C07270=1062.569,160.981,-81.280,172.441,30.431,155.615
C07271=1062.574,161.230,-81.303,172.443,30.435,155.616
C07272=1062.579,161.479,-81.325,172.445,30.437,155.616
C07273=1062.585,161.728,-81.347,172.446,30.440,155.616
C07274=1062.591,161.977,-81.369,172.448,30.443,155.617
C07275=1062.596,162.226,-81.392,172.450,30.446,155.617
C07276=1062.602,162.475,-81.413,172.453,30.449,155.618
C07277=1062.608,162.724,-81.436,172.454,30.452,155.618
C07278=1062.613,162.973,-81.458,172.456,30.455,155.619
C07279=1062.619,163.222,-81.480,172.458,30.458,155.619
C07280=1062.624,163.471,-81.503,172.460,30.461,155.620
C07281=1062.630,163.720,-81.525,172.461,30.463,155.620
C07282=1062.636,163.968,-81.547,172.463,30.466,155.621
C07283=1062.641,164.217,-81.569,172.465,30.469,155.621
C07284=1062.647,164.466,-81.592,172.468,30.472,155.622
C07285=1062.653,164.716,-81.614,172.469,30.475,155.622
C07286=1062.658,164.964,-81.636,172.471,30.478,155.622
C07287=1062.664,165.213,-81.659,172.473,30.481,155.623
C07288=1062.670,165.462,-81.681,172.475,30.484,155.623
C07289=1062.675,165.711,-81.703,172.476,30.487,155.624
C07290=1062.681,165.960,-81.726,172.478,30.490,155.624
C07291=1062.687,166.209,-81.747,172.480,30.492,155.625
C07292=1062.693,166.458,-81.770,172.483,30.496,155.625
C07293=1062.698,166.707,-81.793,172.484,30.498,155.626
C07294=1062.704,166.956,-81.815,172.486,30.501,155.626
C07295=1062.710,167.204,-81.837,172.488,30.504,155.627
C07296=1062.715,167.454,-81.860,172.490,30.507,155.627
C07297=1062.721,167.702,-81.883,172.491,30.510,155.627
C07298=1062.727,167.952,-81.904,172.494,30.513,155.628
C07299=1062.733,168.201,-81.927,172.496,30.516,155.628
C07300=1062.738,168.449,-81.950,172.498,30.519,155.629
C07301=1062.743,168.698,-81.972,172.499,30.521,155.629
C07302=1062.750,168.947,-81.994,172.501,30.524,155.630
C07303=1062.755,169.196,-82.017,172.503,30.527,155.630
C07304=1062.761,169.445,-82.040,172.506,30.530,155.631
C07305=1062.767,169.694,-82.062,172.507,30.533,155.631
C07306=1062.773,169.943,-82.084,172.509,30.536,155.632
C07307=1062.778,170.192,-82.107,172.511,30.539,155.632
C07308=1062.784,170.440,-82.130,172.513,30.541,155.632
C07309=1062.790,170.689,-82.152,172.514,30.545,155.633
C07310=1062.795,170.939,-82.174,172.517,30.547,155.633
C07311=1062.801,171.187,-82.197,172.519,30.551,155.634
C07312=1062.807,171.436,-82.220,172.521,30.553,155.634
C07313=1062.813,171.685,-82.243,172.523,30.556,155.635
C07314=1062.819,171.934,-82.265,172.524,30.559,155.635
C07315=1062.824,172.183,-82.288,172.526,30.562,155.636
C07316=1062.830,172.431,-82.310,172.529,30.565,155.636
C07317=1062.835,172.680,-82.333,172.531,30.568,155.637
C07318=1062.842,172.930,-82.355,172.532,30.571,155.637
C07319=1062.847,173.178,-82.378,172.534,30.573,155.637
C07320=1062.853,173.427,-82.401,172.536,30.576,155.638
C07321=1062.859,173.676,-82.424,172.539,30.579,155.638
C07322=1062.865,173.925,-82.446,172.540,30.582,155.639
C07323=1062.871,174.174,-82.469,172.542,30.585,155.639
C07324=1062.877,174.458,-82.494,172.545,30.589,155.640
C07325=1062.884,174.741,-82.521,172.547,30.592,155.640
C07326=1062.891,175.024,-82.547,172.549,30.595,155.641
C07327=1062.897,175.308,-82.572,172.551,30.598,155.641
C07328=1062.903,175.557,-82.595,172.553,30.601,155.642
C07329=1062.909,175.806,-82.618,172.556,30.604,155.642
C07330=1062.914,176.055,-82.641,172.557,30.607,155.643
C07331=1062.920,176.304,-82.664,172.559,30.610,155.643
C07332=1062.927,176.552,-82.686,172.561,30.612,155.644
C07333=1062.932,176.801,-82.709,172.564,30.616,155.644
C07334=1062.938,177.050,-82.732,172.565,30.618,155.645
C07335=1062.944,177.299,-82.755,172.567,30.621,155.645
C07336=1062.950,177.548,-82.778,172.569,30.624,155.646
C07337=1062.956,177.797,-82.800,172.572,30.627,155.646
C07338=1062.962,178.045,-82.823,172.573,30.630,155.646
C07339=1062.968,178.294,-82.846,172.575,30.633,155.647
C07340=1062.974,178.544,-82.869,172.577,30.636,155.647
C07341=1062.980,178.793,-82.892,172.580,30.638,155.648
C07342=1062.985,179.042,-82.915,172.581,30.642,155.648
C07343=1062.991,179.291,-82.938,172.583,30.644,155.649
C07344=1062.997,179.539,-82.961,172.585,30.647,155.649
C07345=1063.003,179.788,-82.984,172.588,30.650,155.650
C07346=1063.009,180.037,-83.007,172.590,30.653,155.650
C07347=1063.015,180.286,-83.029,172.591,30.656,155.651
C07348=1063.020,180.535,-83.052,172.593,30.659,155.651
C07349=1063.026,180.784,-83.075,172.596,30.662,155.651
C07350=1063.033,181.033,-83.099,172.598,30.665,155.652
C07351=1063.039,181.281,-83.122,172.599,30.667,155.652
C07352=1063.045,181.530,-83.145,172.601,30.670,155.653
C07353=1063.051,181.779,-83.168,172.604,30.673,155.653
C07354=1063.056,182.028,-83.191,172.606,30.676,155.654
C07355=1063.062,182.277,-83.214,172.607,30.679,155.654
C07356=1063.068,182.526,-83.236,172.610,30.682,155.655
C07357=1063.075,182.775,-83.261,172.612,30.685,155.655
C07358=1063.080,183.024,-83.283,172.614,30.687,155.655
C07359=1063.087,183.272,-83.306,172.615,30.691,155.656
C07360=1063.092,183.521,-83.329,172.618,30.693,155.656
C07361=1063.099,183.769,-83.352,172.620,30.696,155.657
C07362=1063.105,184.019,-83.376,172.622,30.699,155.657
C07363=1063.111,184.268,-83.399,172.625,30.702,155.658
C07364=1063.116,184.517,-83.422,172.626,30.705,155.658
C07365=1063.122,184.765,-83.445,172.628,30.708,155.659
C07366=1063.127,185.014,-83.469,172.631,30.711,155.659
C07367=1063.133,185.263,-83.492,172.633,30.714,155.660
C07368=1063.139,185.511,-83.515,172.634,30.717,155.660
C07369=1063.144,185.761,-83.539,172.636,30.720,155.661
C07370=1063.150,186.010,-83.562,172.639,30.723,155.661
C07371=1063.156,186.258,-83.586,172.641,30.726,155.662
C07372=1063.161,186.508,-83.609,172.642,30.730,155.662
C07373=1063.168,186.756,-83.633,172.645,30.732,155.663
C07374=1063.172,187.005,-83.657,172.647,30.736,155.663
C07375=1063.178,187.254,-83.680,172.649,30.739,155.664
C07376=1063.184,187.502,-83.703,172.650,30.742,155.664
C07377=1063.189,187.752,-83.727,172.653,30.745,155.665
C07378=1063.195,188.000,-83.750,172.655,30.748,155.665
C07379=1063.202,188.249,-83.774,172.657,30.751,155.666
C07380=1063.207,188.498,-83.798,172.659,30.754,155.666
C07381=1063.213,188.747,-83.821,172.661,30.757,155.666
C07382=1063.218,188.996,-83.845,172.663,30.760,155.667
C07383=1063.224,189.244,-83.868,172.666,30.763,155.667
C07384=1063.230,189.493,-83.892,172.668,30.766,155.668
C07385=1063.235,189.743,-83.916,172.669,30.769,155.668
C07386=1063.241,189.991,-83.939,172.672,30.773,155.669
C07387=1063.247,190.239,-83.964,172.674,30.775,155.669
C07388=1063.253,190.523,-83.990,172.677,30.779,155.670
C07389=1063.260,190.806,-84.017,172.678,30.782,155.671
C07390=1063.267,191.089,-84.043,172.681,30.786,155.671
C07391=1063.273,191.372,-84.071,172.684,30.789,155.672
C07392=1063.279,191.620,-84.094,172.686,30.792,155.672
C07393=1063.284,191.870,-84.118,172.687,30.795,155.673
C07394=1063.290,192.118,-84.142,172.690,30.798,155.673
C07395=1063.296,192.367,-84.166,172.692,30.801,155.674
C07396=1063.301,192.616,-84.189,172.694,30.805,155.674
C07397=1063.308,192.865,-84.213,172.696,30.807,155.675
C07398=1063.313,193.114,-84.238,172.698,30.811,155.675
C07399=1063.319,193.362,-84.260,172.700,30.814,155.676
C07400=1063.325,193.612,-84.285,172.703,30.817,155.676
C07401=1063.331,193.860,-84.309,172.704,30.820,155.677
C07402=1063.336,194.109,-84.332,172.707,30.823,155.677
C07403=1063.342,194.357,-84.356,172.709,30.826,155.678
C07404=1063.348,194.607,-84.381,172.711,30.829,155.678
C07405=1063.354,194.855,-84.404,172.714,30.832,155.679
C07406=1063.359,195.104,-84.428,172.715,30.835,155.679
C07407=1063.366,195.353,-84.452,172.717,30.838,155.680
C07408=1063.372,195.601,-84.475,172.720,30.842,155.680
C07409=1063.377,195.850,-84.500,172.722,30.844,155.680
C07410=1063.384,196.099,-84.524,172.724,30.848,155.681
C07411=1063.389,196.348,-84.547,172.726,30.851,155.682
C07412=1063.395,196.597,-84.571,172.728,30.853,155.682
C07413=1063.401,196.846,-84.596,172.731,30.857,155.682
C07414=1063.407,197.094,-84.619,172.732,30.860,155.683
C07415=1063.412,197.343,-84.643,172.735,30.863,155.683
C07416=1063.419,197.592,-84.668,172.737,30.866,155.684
C07417=1063.424,197.840,-84.692,172.739,30.869,155.684
C07418=1063.430,198.089,-84.716,172.742,30.872,155.685
C07419=1063.435,198.338,-84.739,172.743,30.875,155.685
C07420=1063.441,198.587,-84.763,172.746,30.879,155.686
C07421=1063.447,198.836,-84.788,172.748,30.881,155.686
C07422=1063.453,199.084,-84.811,172.751,30.884,155.687
C07423=1063.459,199.334,-84.836,172.752,30.888,155.687
C07424=1063.465,199.582,-84.860,172.754,30.891,155.688
C07425=1063.471,199.831,-84.884,172.757,30.894,155.688
C07426=1063.477,200.079,-84.908,172.759,30.897,155.689
C07427=1063.483,200.328,-84.932,172.761,30.900,155.689
C07428=1063.489,200.577,-84.956,172.763,30.903,155.690
C07429=1063.495,200.826,-84.980,172.766,30.906,155.690
C07430=1063.500,201.075,-85.005,172.768,30.909,155.691
C07431=1063.506,201.323,-85.029,172.770,30.912,155.691
C07432=1063.512,201.572,-85.053,172.772,30.915,155.692
C07433=1063.518,201.821,-85.077,172.774,30.919,155.692
C07434=1063.524,202.070,-85.102,172.777,30.921,155.693
C07435=1063.530,202.318,-85.125,172.779,30.925,155.693
C07436=1063.537,202.567,-85.151,172.781,30.928,155.694
C07437=1063.542,202.816,-85.175,172.783,30.931,155.694
C07438=1063.548,203.065,-85.199,172.786,30.934,155.695
C07439=1063.553,203.313,-85.224,172.788,30.938,155.695
C07440=1063.559,203.562,-85.247,172.790,30.941,155.696
C07441=1063.565,203.811,-85.272,172.792,30.944,155.697
C07442=1063.571,204.059,-85.297,172.794,30.947,155.697
C07443=1063.576,204.308,-85.322,172.797,30.950,155.697
C07444=1063.582,204.557,-85.346,172.799,30.953,155.698
C07445=1063.588,204.806,-85.370,172.801,30.957,155.699
C07446=1063.594,205.054,-85.394,172.803,30.960,155.699
C07447=1063.600,205.303,-85.419,172.806,30.963,155.700
C07448=1063.605,205.552,-85.444,172.808,30.966,155.700
C07449=1063.611,205.801,-85.468,172.811,30.970,155.701
C07450=1063.617,206.049,-85.493,172.812,30.973,155.701
C07451=1063.623,206.298,-85.518,172.815,30.976,155.702
C07452=1063.647,207.346,-85.621,172.981,31.057,155.708
C07453=1063.653,207.569,-85.644,172.982,31.060,155.709
C07454=1063.659,207.793,-85.667,172.984,31.064,155.710
C07455=1063.664,208.016,-85.689,172.986,31.068,155.710
C07456=1063.669,208.240,-85.712,172.988,31.071,155.711
C07457=1063.675,208.463,-85.735,172.988,31.075,155.712
C07458=1063.680,208.688,-85.758,172.990,31.079,155.712
C07459=1063.685,208.910,-85.781,172.992,31.082,155.713
C07460=1063.691,209.134,-85.804,172.994,31.086,155.714
C07461=1063.697,209.383,-85.829,172.996,31.090,155.714
C07462=1063.703,209.631,-85.854,172.998,31.094,155.715
C07463=1063.709,209.880,-85.880,173.000,31.098,155.716
C07464=1063.715,210.129,-85.906,173.002,31.102,155.717
C07465=1063.721,210.378,-85.931,173.004,31.106,155.717
C07466=1063.728,210.626,-85.957,173.006,31.111,155.718
C07467=1063.733,210.875,-85.983,173.008,31.114,155.719
C07468=1063.739,211.123,-86.008,173.010,31.119,155.720
C07469=1063.745,211.372,-86.034,173.012,31.122,155.720
C07470=1063.752,211.621,-86.059,173.014,31.127,155.721
C07471=1063.757,211.869,-86.085,173.016,31.131,155.722
C07472=1063.763,212.117,-86.111,173.018,31.135,155.722
C07473=1063.769,212.366,-86.136,173.020,31.139,155.723
C07474=1063.775,212.615,-86.162,173.022,31.143,155.724
C07475=1063.781,212.863,-86.187,173.024,31.147,155.725
C07476=1063.787,213.112,-86.213,173.026,31.151,155.725
C07477=1063.793,213.360,-86.239,173.027,31.155,155.726
C07478=1063.799,213.609,-86.265,173.030,31.159,155.727
C07479=1063.805,213.858,-86.290,173.032,31.164,155.728
C07480=1063.811,214.106,-86.317,173.034,31.167,155.728
C07481=1063.817,214.355,-86.342,173.036,31.172,155.729
C07482=1063.823,214.604,-86.368,173.037,31.175,155.730
C07483=1063.829,214.852,-86.393,173.040,31.180,155.730
C07484=1063.835,215.101,-86.420,173.042,31.184,155.731
C07485=1063.841,215.349,-86.445,173.044,31.188,155.732
C07486=1063.847,215.598,-86.472,173.045,31.192,155.733
C07487=1063.853,215.846,-86.497,173.048,31.196,155.733
C07488=1063.858,216.095,-86.523,173.050,31.200,155.734
C07489=1063.865,216.343,-86.549,173.052,31.204,155.735
C07490=1063.871,216.592,-86.574,173.054,31.208,155.736
C07491=1063.877,216.840,-86.601,173.056,31.212,155.736
C07492=1063.884,217.090,-86.627,173.058,31.216,155.737
C07493=1063.889,217.339,-86.653,173.060,31.220,155.738
C07494=1063.896,217.587,-86.679,173.062,31.225,155.738
C07495=1063.901,217.836,-86.705,173.064,31.228,155.739
C07496=1063.908,218.084,-86.731,173.066,31.233,155.740
C07497=1063.913,218.333,-86.757,173.068,31.236,155.741
C07498=1063.920,218.581,-86.783,173.070,31.240,155.741
C07499=1063.925,218.830,-86.809,173.072,31.244,155.742
C07500=1063.932,219.078,-86.835,173.074,31.248,155.743
C07501=1063.937,219.327,-86.861,173.077,31.253,155.743
C07502=1063.944,219.576,-86.887,173.079,31.256,155.744
C07503=1063.950,219.825,-86.913,173.080,31.261,155.745
C07504=1063.956,220.073,-86.939,173.083,31.264,155.746
C07505=1063.962,220.321,-86.966,173.085,31.268,155.746
C07506=1063.968,220.570,-86.991,173.087,31.272,155.747
C07507=1063.974,220.818,-87.018,173.088,31.276,155.748
C07508=1063.980,221.067,-87.043,173.091,31.281,155.748
C07509=1063.985,221.293,-87.067,173.093,31.284,155.749
C07510=1063.991,221.519,-87.091,173.095,31.287,155.750
C07511=1063.996,221.745,-87.115,173.097,31.291,155.750
C07512=1064.002,221.971,-87.139,173.098,31.295,155.751
C07513=1064.008,222.197,-87.163,173.100,31.299,155.752
C07514=1064.013,222.423,-87.187,173.102,31.302,155.752
C07515=1064.019,222.649,-87.211,173.104,31.306,155.753
C07516=1064.023,222.875,-87.235,173.106,31.310,155.754
C07517=1064.030,223.124,-87.262,173.108,31.314,155.754
C07518=1064.036,223.372,-87.288,173.110,31.318,155.755
C07519=1064.042,223.621,-87.314,173.112,31.322,155.756
C07520=1064.047,223.869,-87.340,173.115,31.326,155.757
C07521=1064.053,224.118,-87.367,173.116,31.330,155.757
C07522=1064.060,224.366,-87.393,173.118,31.334,155.758
C07523=1064.066,224.615,-87.420,173.121,31.338,155.759
C07524=1064.072,224.864,-87.446,173.123,31.342,155.759
C07525=1064.077,225.112,-87.473,173.125,31.346,155.760
C07526=1064.084,225.360,-87.499,173.127,31.350,155.761
C07527=1064.090,225.608,-87.525,173.129,31.354,155.762
C07528=1064.096,225.857,-87.552,173.131,31.358,155.762
C07529=1064.102,226.106,-87.579,173.134,31.362,155.763
C07530=1064.107,226.355,-87.605,173.135,31.366,155.764
C07531=1064.114,226.603,-87.631,173.137,31.370,155.764
C07532=1064.120,226.852,-87.658,173.140,31.374,155.765
C07533=1064.126,227.100,-87.685,173.142,31.378,155.766
C07534=1064.132,227.349,-87.711,173.145,31.382,155.767
C07535=1064.137,227.597,-87.738,173.146,31.386,155.767
C07536=1064.145,227.846,-87.764,173.148,31.390,155.768
C07537=1064.150,228.094,-87.791,173.151,31.394,155.769
C07538=1064.156,228.342,-87.818,173.153,31.398,155.769
C07539=1064.163,228.592,-87.845,173.154,31.402,155.770
C07540=1064.168,228.840,-87.871,173.157,31.406,155.771
C07541=1064.175,229.088,-87.898,173.159,31.409,155.772
C07542=1064.181,229.337,-87.925,173.161,31.414,155.772
C07543=1064.187,229.585,-87.951,173.164,31.417,155.773
C07544=1064.193,229.834,-87.978,173.165,31.422,155.774
C07545=1064.199,230.083,-88.005,173.168,31.426,155.774
C07546=1064.205,230.331,-88.031,173.170,31.429,155.775
C07547=1064.211,230.580,-88.058,173.172,31.434,155.776
C07548=1064.216,230.828,-88.085,173.175,31.437,155.777
C07549=1064.223,231.076,-88.113,173.176,31.442,155.777
C07550=1064.229,231.325,-88.139,173.179,31.445,155.778
C07551=1064.235,231.573,-88.166,173.181,31.450,155.779
C07552=1064.241,231.822,-88.193,173.183,31.453,155.779
C07553=1064.247,232.070,-88.219,173.186,31.457,155.780
C07554=1064.253,232.319,-88.246,173.187,31.462,155.781
C07555=1064.259,232.567,-88.274,173.189,31.465,155.782
C07556=1064.265,232.816,-88.300,173.192,31.470,155.782
C07557=1064.271,233.064,-88.327,173.194,31.473,155.783
C07558=1064.277,233.313,-88.354,173.197,31.477,155.784
C07559=1064.283,233.561,-88.381,173.198,31.481,155.784
C07560=1064.289,233.810,-88.409,173.200,31.485,155.785
C07561=1064.295,234.059,-88.436,173.203,31.490,155.786
C07562=1064.300,234.307,-88.462,173.205,31.493,155.787
C07563=1064.307,234.555,-88.490,173.208,31.498,155.787
C07564=1064.313,234.804,-88.517,173.209,31.501,155.788
C07565=1064.318,235.026,-88.541,173.211,31.505,155.789
C07566=1064.323,235.248,-88.565,173.213,31.508,155.789
C07567=1064.329,235.470,-88.590,173.216,31.512,155.790
C07568=1064.334,235.691,-88.614,173.218,31.516,155.791
C07569=1064.340,235.914,-88.638,173.219,31.519,155.791
C07570=1064.345,236.136,-88.663,173.221,31.523,155.792
C07571=1064.351,236.358,-88.687,173.223,31.526,155.792
C07572=1064.356,236.580,-88.711,173.225,31.530,155.793
C07573=1064.361,236.828,-88.738,173.228,31.534,155.794
C07574=1064.368,237.077,-88.765,173.230,31.538,155.795
C07575=1064.374,237.325,-88.793,173.232,31.542,155.795
C07576=1064.380,237.574,-88.820,173.234,31.545,155.796
C07577=1064.386,237.822,-88.847,173.237,31.550,155.797
C07578=1064.392,238.071,-88.874,173.239,31.554,155.797
C07579=1064.398,238.319,-88.902,173.242,31.557,155.798
C07580=1064.404,238.568,-88.929,173.243,31.562,155.799
C07581=1064.410,238.816,-88.956,173.245,31.565,155.800
C07582=1064.416,239.065,-88.984,173.248,31.569,155.800
C07583=1064.422,239.313,-89.011,173.250,31.573,155.801
C07584=1064.429,239.562,-89.038,173.253,31.577,155.802
C07585=1064.435,239.809,-89.066,173.254,31.581,155.802
C07586=1064.441,240.058,-89.094,173.257,31.585,155.803
C07587=1064.446,240.307,-89.121,173.259,31.589,155.804
C07588=1064.453,240.555,-89.148,173.262,31.593,155.805
C07589=1064.458,240.804,-89.176,173.264,31.597,155.805
C07590=1064.465,241.052,-89.203,173.267,31.601,155.806
C07591=1064.471,241.300,-89.231,173.268,31.605,155.807
C07592=1064.477,241.549,-89.258,173.271,31.609,155.807
C07593=1064.483,241.797,-89.286,173.273,31.613,155.808
C07594=1064.489,242.045,-89.313,173.276,31.617,155.809
C07595=1064.495,242.294,-89.340,173.278,31.621,155.809
C07596=1064.501,242.542,-89.368,173.280,31.625,155.810
C07597=1064.508,242.791,-89.396,173.282,31.629,155.811
C07598=1064.513,243.040,-89.423,173.284,31.632,155.812
C07599=1064.519,243.288,-89.451,173.287,31.636,155.812
C07600=1064.525,243.536,-89.479,173.289,31.641,155.813
C07601=1064.531,243.785,-89.507,173.292,31.644,155.814
C07602=1064.537,244.033,-89.535,173.293,31.649,155.815
C07603=1064.543,244.282,-89.562,173.296,31.652,155.815
C07604=1064.548,244.530,-89.590,173.298,31.657,155.816
C07605=1064.555,244.778,-89.617,173.301,31.660,155.817
C07606=1064.560,245.026,-89.645,173.303,31.664,155.817
C07607=1064.567,245.275,-89.673,173.305,31.669,155.818
C07608=1064.573,245.523,-89.701,173.307,31.672,155.819
C07609=1064.579,245.771,-89.729,173.310,31.676,155.819
C07610=1064.585,246.021,-89.756,173.312,31.680,155.820
C07611=1064.591,246.268,-89.784,173.315,31.684,155.821
C07612=1064.597,246.517,-89.812,173.317,31.688,155.822
C07613=1064.603,246.766,-89.840,173.319,31.692,155.822
C07614=1064.609,247.013,-89.868,173.322,31.696,155.823
C07615=1064.615,247.262,-89.896,173.324,31.700,155.824
C07616=1064.620,247.510,-89.924,173.327,31.704,155.824
C07617=1064.626,247.759,-89.952,173.329,31.708,155.825
C07618=1064.633,248.007,-89.980,173.332,31.712,155.826
C07619=1064.638,248.256,-90.008,173.333,31.716,155.827
C07620=1064.644,248.504,-90.036,173.336,31.720,155.827
C07621=1064.649,248.723,-90.061,173.338,31.724,155.828
C07622=1064.654,248.942,-90.086,173.340,31.727,155.829
C07623=1064.660,249.161,-90.111,173.342,31.731,155.829
C07624=1064.665,249.380,-90.136,173.345,31.734,155.830
C07625=1064.670,249.599,-90.160,173.346,31.738,155.831
C07626=1064.675,249.818,-90.185,173.348,31.741,155.831
C07627=1064.681,250.036,-90.210,173.350,31.745,155.832
C07628=1064.686,250.255,-90.235,173.352,31.748,155.833
C07629=1064.692,250.502,-90.263,173.355,31.752,155.833
C07630=1064.698,250.751,-90.291,173.358,31.757,155.834
C07631=1064.704,251.000,-90.319,173.360,31.760,155.835
C07632=1064.709,251.248,-90.347,173.362,31.764,155.835
C07633=1064.715,251.497,-90.376,173.364,31.768,155.836
C07634=1064.722,251.745,-90.403,173.367,31.772,155.837
C07635=1064.728,251.993,-90.432,173.369,31.776,155.838
C07636=1064.734,252.241,-90.460,173.372,31.780,155.838
C07637=1064.739,252.490,-90.489,173.375,31.784,155.839
C07638=1064.745,252.739,-90.517,173.376,31.788,155.840
C07639=1064.752,252.986,-90.545,173.379,31.792,155.840
C07640=1064.758,253.235,-90.573,173.381,31.796,155.841
C07641=1064.764,253.483,-90.602,173.384,31.800,155.842
C07642=1064.770,253.732,-90.631,173.386,31.804,155.843
C07643=1064.775,253.980,-90.659,173.389,31.808,155.843
C07644=1064.782,254.228,-90.687,173.391,31.812,155.844
C07645=1064.788,254.476,-90.716,173.393,31.816,155.845
C07646=1064.794,254.725,-90.744,173.396,31.820,155.845
C07647=1064.800,254.973,-90.772,173.398,31.823,155.846
C07648=1064.806,255.221,-90.801,173.401,31.828,155.847
C07649=1064.812,255.470,-90.829,173.404,31.832,155.848
C07650=1064.819,255.718,-90.858,173.406,31.835,155.848
C07651=1064.825,255.966,-90.886,173.408,31.840,155.849
C07652=1064.830,256.214,-90.915,173.410,31.843,155.850
C07653=1064.836,256.463,-90.943,173.413,31.847,155.850
C07654=1064.842,256.711,-90.971,173.416,31.851,155.851
C07655=1064.848,256.960,-91.000,173.418,31.855,155.852
C07656=1064.854,257.208,-91.029,173.421,31.859,155.853
C07657=1064.861,257.456,-91.057,173.422,31.863,155.853
C07658=1064.867,257.705,-91.085,173.425,31.867,155.854
C07659=1064.873,257.952,-91.114,173.428,31.871,155.855
C07660=1064.879,258.200,-91.143,173.430,31.875,155.855
C07661=1064.885,258.449,-91.171,173.433,31.879,155.856
C07662=1064.891,258.697,-91.201,173.436,31.883,155.857
C07663=1064.897,258.946,-91.229,173.438,31.887,155.858
C07664=1064.904,259.194,-91.258,173.440,31.891,155.858
C07665=1064.910,259.443,-91.286,173.443,31.894,155.859
C07666=1064.917,259.691,-91.315,173.445,31.898,155.860
C07667=1064.923,259.939,-91.344,173.448,31.902,155.860
C07668=1064.929,260.188,-91.372,173.450,31.906,155.861
C07669=1064.935,260.436,-91.401,173.453,31.910,155.862
C07670=1064.941,260.684,-91.430,173.456,31.914,155.863
C07671=1064.947,260.932,-91.458,173.457,31.918,155.863
C07672=1064.953,261.180,-91.487,173.460,31.922,155.864
C07673=1064.959,261.428,-91.516,173.463,31.926,155.865
C07674=1064.965,261.676,-91.545,173.465,31.929,155.865
C07675=1064.971,261.925,-91.574,173.468,31.933,155.866
C07676=1064.977,262.173,-91.603,173.471,31.938,155.867
C07677=1064.984,262.391,-91.627,173.473,31.941,155.867
C07678=1064.989,262.609,-91.653,173.475,31.944,155.868
C07679=1064.994,262.827,-91.678,173.477,31.948,155.869
C07680=1065.000,263.045,-91.704,173.479,31.951,155.869
C07681=1065.006,263.262,-91.729,173.482,31.954,155.870
C07682=1065.011,263.480,-91.754,173.484,31.958,155.871
C07683=1065.016,263.698,-91.780,173.486,31.961,155.871
C07684=1065.022,263.915,-91.806,173.489,31.965,155.872
C07685=1065.028,264.164,-91.834,173.491,31.969,155.872
C07686=1065.033,264.412,-91.864,173.493,31.973,155.873
C07687=1065.040,264.661,-91.893,173.496,31.977,155.874
C07688=1065.045,264.908,-91.921,173.498,31.981,155.875
C07689=1065.052,265.156,-91.950,173.501,31.985,155.875
C07690=1065.057,265.405,-91.980,173.504,31.989,155.876
C07691=1065.063,265.653,-92.009,173.506,31.993,155.877
C07692=1065.070,265.901,-92.038,173.509,31.996,155.878
C07693=1065.076,266.149,-92.067,173.511,32.001,155.878
C07694=1065.081,266.397,-92.097,173.514,32.005,155.879
C07695=1065.088,266.645,-92.126,173.516,32.009,155.880
C07696=1065.094,266.894,-92.155,173.519,32.012,155.880
C07697=1065.100,267.143,-92.185,173.522,32.017,155.881
C07698=1065.106,267.391,-92.214,173.524,32.020,155.882
C07699=1065.112,267.639,-92.243,173.527,32.024,155.883
C07700=1065.119,267.887,-92.273,173.530,32.029,155.883
C07701=1065.125,268.135,-92.302,173.531,32.032,155.884
C07702=1065.131,268.383,-92.331,173.534,32.037,155.885
C07703=1065.137,268.631,-92.360,173.537,32.040,155.886
C07704=1065.143,268.880,-92.390,173.540,32.044,155.886
C07705=1065.149,269.128,-92.419,173.542,32.048,155.887
C07706=1065.155,269.376,-92.448,173.545,32.052,155.888
C07707=1065.161,269.624,-92.479,173.548,32.056,155.888
C07708=1065.167,269.872,-92.508,173.551,32.060,155.889
C07709=1065.173,270.120,-92.537,173.552,32.064,155.890
C07710=1065.179,270.369,-92.567,173.555,32.068,155.891
C07711=1065.185,270.617,-92.597,173.558,32.072,155.891
C07712=1065.192,270.865,-92.626,173.561,32.076,155.892
C07713=1065.198,271.113,-92.655,173.563,32.080,155.893
C07714=1065.203,271.362,-92.685,173.566,32.084,155.894
C07715=1065.210,271.609,-92.714,173.569,32.088,155.894
C07716=1065.215,271.858,-92.744,173.572,32.092,155.895
C07717=1065.222,272.105,-92.774,173.573,32.096,155.896
C07718=1065.228,272.354,-92.804,173.576,32.100,155.897
C07719=1065.234,272.602,-92.833,173.579,32.104,155.897
C07720=1065.240,272.850,-92.863,173.582,32.108,155.898
C07721=1065.246,273.098,-92.892,173.584,32.112,155.899
C07722=1065.252,273.347,-92.922,173.587,32.116,155.899
C07723=1065.258,273.594,-92.952,173.590,32.120,155.900
C07724=1065.264,273.843,-92.981,173.593,32.124,155.901
C07725=1065.271,274.091,-93.011,173.594,32.128,155.902
C07726=1065.277,274.339,-93.041,173.597,32.132,155.902
C07727=1065.282,274.587,-93.071,173.600,32.136,155.903
C07728=1065.289,274.835,-93.100,173.603,32.140,155.904
C07729=1065.294,275.083,-93.131,173.606,32.144,155.905
C07730=1065.301,275.332,-93.160,173.608,32.148,155.905
C07731=1065.307,275.580,-93.191,173.611,32.152,155.906
C07732=1065.313,275.828,-93.221,173.614,32.156,155.907
C07733=1065.318,276.048,-93.247,173.616,32.160,155.908
C07734=1065.323,276.267,-93.273,173.618,32.163,155.908
C07735=1065.329,276.487,-93.300,173.620,32.167,155.909
C07736=1065.335,276.706,-93.326,173.623,32.170,155.909
C07737=1065.340,276.925,-93.353,173.625,32.174,155.910
C07738=1065.346,277.145,-93.379,173.628,32.178,155.911
C07739=1065.350,277.364,-93.406,173.630,32.181,155.911
C07740=1065.356,277.584,-93.433,173.633,32.185,155.912
C07741=1065.362,277.832,-93.462,173.636,32.189,155.913
C07742=1065.368,278.080,-93.493,173.638,32.192,155.914
C07743=1065.374,278.328,-93.523,173.641,32.197,155.914
C07744=1065.380,278.577,-93.553,173.643,32.201,155.915
C07745=1065.387,278.825,-93.583,173.646,32.205,155.916
C07746=1065.393,279.073,-93.613,173.649,32.209,155.916
C07747=1065.399,279.321,-93.644,173.651,32.213,155.917
C07748=1065.405,279.569,-93.673,173.654,32.217,155.918
C07749=1065.411,279.817,-93.703,173.657,32.221,155.919
C07750=1065.417,280.066,-93.734,173.660,32.225,155.920
C07751=1065.423,280.313,-93.764,173.663,32.229,155.920
C07752=1065.429,280.561,-93.795,173.666,32.233,155.921
C07753=1065.436,280.809,-93.824,173.667,32.237,155.922
C07754=1065.442,281.058,-93.854,173.670,32.241,155.923
C07755=1065.448,281.306,-93.885,173.673,32.245,155.923
C07756=1065.453,281.553,-93.915,173.676,32.249,155.924
C07757=1065.460,281.802,-93.946,173.679,32.253,155.925
C07758=1065.466,282.050,-93.976,173.682,32.258,155.926
C07759=1065.471,282.298,-94.007,173.684,32.261,155.926
C07760=1065.478,282.546,-94.037,173.687,32.266,155.927
C07761=1065.484,282.794,-94.068,173.690,32.269,155.928
C07762=1065.489,283.042,-94.098,173.693,32.274,155.929
C07763=1065.496,283.290,-94.129,173.695,32.278,155.929
C07764=1065.502,283.538,-94.159,173.698,32.282,155.930
C07765=1065.508,283.786,-94.189,173.701,32.286,155.931
C07766=1065.514,284.034,-94.220,173.704,32.290,155.932
C07767=1065.520,284.282,-94.250,173.706,32.294,155.932
C07768=1065.526,284.531,-94.281,173.709,32.298,155.933
C07769=1065.532,284.778,-94.312,173.712,32.302,155.934
C07770=1065.539,285.026,-94.342,173.715,32.306,155.935
C07771=1065.545,285.274,-94.373,173.718,32.310,155.935
C07772=1065.551,285.522,-94.403,173.721,32.314,155.936
C07773=1065.558,285.770,-94.434,173.724,32.318,155.937
C07774=1065.563,286.018,-94.464,173.726,32.323,155.938
C07775=1065.570,286.266,-94.496,173.728,32.326,155.938
C07776=1065.576,286.514,-94.526,173.731,32.331,155.939
C07777=1065.582,286.762,-94.556,173.734,32.335,155.940
C07778=1065.588,287.010,-94.587,173.737,32.339,155.941
C07779=1065.594,287.258,-94.617,173.740,32.343,155.941
C07780=1065.601,287.506,-94.649,173.743,32.347,155.942
C07781=1065.606,287.754,-94.679,173.746,32.351,155.943
C07782=1065.613,288.002,-94.710,173.749,32.355,155.944
C07783=1065.619,288.250,-94.741,173.752,32.359,155.945
C07784=1065.625,288.498,-94.772,173.755,32.363,155.945
C07785=1065.631,288.746,-94.803,173.757,32.367,155.946
C07786=1065.637,288.994,-94.834,173.760,32.372,155.947
C07787=1065.643,289.242,-94.864,173.762,32.375,155.947
C07788=1065.649,289.490,-94.895,173.765,32.380,155.948
C07789=1065.654,289.715,-94.923,173.768,32.383,155.949
C07790=1065.661,289.940,-94.951,173.771,32.387,155.950
C07791=1065.666,290.165,-94.980,173.773,32.391,155.950
C07792=1065.672,290.389,-95.007,173.776,32.394,155.951
C07793=1065.677,290.614,-95.036,173.779,32.399,155.952
C07794=1065.683,290.839,-95.064,173.781,32.402,155.953
C07795=1065.688,291.063,-95.092,173.784,32.406,155.953
C07796=1065.694,291.288,-95.121,173.787,32.410,155.954
C07797=1065.700,291.536,-95.151,173.789,32.414,155.955
C07798=1065.706,291.784,-95.182,173.792,32.418,155.955
C07799=1065.712,292.032,-95.213,173.795,32.422,155.956
C07800=1065.718,292.280,-95.245,173.798,32.426,155.957
C07801=1065.725,292.529,-95.276,173.801,32.430,155.958
C07802=1065.731,292.776,-95.307,173.803,32.435,155.959
C07803=1065.737,293.024,-95.339,173.806,32.438,155.959
C07804=1065.743,293.272,-95.369,173.809,32.443,155.960
C07805=1065.749,293.520,-95.400,173.812,32.447,155.961
C07806=1065.755,293.768,-95.432,173.815,32.451,155.962
C07807=1065.761,294.016,-95.463,173.818,32.455,155.962
C07808=1065.768,294.264,-95.494,173.821,32.459,155.963
C07809=1065.774,294.511,-95.525,173.824,32.463,155.964
C07810=1065.780,294.760,-95.557,173.827,32.468,155.965
C07811=1065.786,295.008,-95.588,173.829,32.472,155.966
C07812=1065.792,295.255,-95.620,173.832,32.476,155.966
C07813=1065.799,295.503,-95.651,173.835,32.480,155.967
C07814=1065.805,295.752,-95.682,173.838,32.484,155.968
C07815=1065.810,295.999,-95.714,173.841,32.488,155.969
C07816=1065.817,296.247,-95.745,173.844,32.493,155.969
C07817=1065.823,296.495,-95.777,173.847,32.497,155.970
C07818=1065.829,296.742,-95.808,173.850,32.501,155.971
C07819=1065.835,296.991,-95.840,173.853,32.505,155.972
C07820=1065.842,297.239,-95.871,173.856,32.510,155.973
C07821=1065.847,297.487,-95.902,173.859,32.514,155.974
C07822=1065.854,297.735,-95.934,173.862,32.518,155.974
C07823=1065.860,297.983,-95.966,173.865,32.522,155.975
C07824=1065.865,298.230,-95.998,173.868,32.527,155.976
C07825=1065.872,298.478,-96.029,173.871,32.531,155.977
C07826=1065.878,298.726,-96.061,173.873,32.535,155.978
C07827=1065.883,298.974,-96.093,173.876,32.539,155.978
C07828=1065.889,299.222,-96.125,173.879,32.544,155.979
C07829=1065.896,299.470,-96.156,173.882,32.548,155.980
C07830=1065.902,299.717,-96.189,173.885,32.552,155.981
C07831=1065.908,299.965,-96.221,173.888,32.556,155.982
C07832=1065.914,300.213,-96.252,173.891,32.561,155.982
C07833=1065.920,300.461,-96.284,173.895,32.565,155.983
C07834=1065.926,300.709,-96.316,173.898,32.569,155.984
C07835=1065.932,300.957,-96.348,173.901,32.574,155.985
C07836=1065.938,301.205,-96.379,173.904,32.578,155.986
C07837=1065.944,301.452,-96.411,173.907,32.583,155.987
C07838=1065.950,301.700,-96.444,173.910,32.587,155.987
C07839=1065.956,301.948,-96.476,173.913,32.591,155.988
C07840=1065.963,302.196,-96.507,173.916,32.595,155.989
C07841=1065.968,302.444,-96.539,173.919,32.600,155.990
C07842=1065.974,302.691,-96.571,173.922,32.604,155.991
C07843=1065.980,302.939,-96.603,173.924,32.608,155.991
C07844=1065.987,303.187,-96.635,173.927,32.612,155.992
C07845=1065.993,303.419,-96.665,173.930,32.617,155.993
C07846=1065.998,303.651,-96.695,173.933,32.620,155.994
C07847=1066.004,303.884,-96.725,173.936,32.624,155.994
C07848=1066.010,304.116,-96.755,173.939,32.629,155.995
C07849=1066.016,304.349,-96.786,173.942,32.632,155.996
C07850=1066.021,304.581,-96.815,173.945,32.637,155.997
C07851=1066.027,304.813,-96.845,173.947,32.641,155.998
C07852=1066.033,305.045,-96.875,173.950,32.644,155.998
C07853=1066.039,305.293,-96.908,173.953,32.649,155.999
C07854=1066.045,305.541,-96.940,173.957,32.654,156.000
C07855=1066.051,305.789,-96.973,173.960,32.658,156.001
C07856=1066.058,306.037,-97.004,173.963,32.662,156.002
C07857=1066.064,306.284,-97.037,173.966,32.666,156.002
C07858=1066.070,306.533,-97.069,173.969,32.670,156.003
C07859=1066.076,306.779,-97.101,173.972,32.675,156.004
C07860=1066.082,307.028,-97.133,173.975,32.679,156.005
C07861=1066.089,307.275,-97.166,173.978,32.683,156.006
C07862=1066.095,307.523,-97.198,173.982,32.688,156.007
C07863=1066.101,307.771,-97.230,173.985,32.692,156.007
C07864=1066.107,308.019,-97.262,173.988,32.697,156.008
C07865=1066.114,308.267,-97.295,173.990,32.701,156.009
C07866=1066.120,308.514,-97.328,173.993,32.705,156.010
C07867=1066.127,308.762,-97.359,173.996,32.709,156.011
C07868=1066.133,309.010,-97.392,173.999,32.713,156.011
C07869=1066.139,309.258,-97.424,174.003,32.718,156.012
C07870=1066.145,309.505,-97.457,174.006,32.723,156.013
C07871=1066.151,309.753,-97.489,174.009,32.727,156.014
C07872=1066.158,310.001,-97.522,174.012,32.731,156.015
C07873=1066.164,310.249,-97.554,174.015,32.735,156.016
C07874=1066.170,310.496,-97.587,174.018,32.740,156.017
C07875=1066.177,310.744,-97.619,174.022,32.744,156.017
C07876=1066.184,310.992,-97.652,174.025,32.749,156.018
C07877=1066.190,311.240,-97.684,174.028,32.753,156.019
C07878=1066.196,311.488,-97.717,174.031,32.757,156.020
C07879=1066.203,311.735,-97.750,174.034,32.761,156.021
C07880=1066.209,311.983,-97.783,174.038,32.766,156.022
C07881=1066.215,312.231,-97.815,174.041,32.770,156.022
C07882=1066.221,312.479,-97.847,174.044,32.775,156.023
C07883=1066.227,312.726,-97.880,174.047,32.779,156.024
C07884=1066.234,312.975,-97.913,174.050,32.783,156.025
C07885=1066.241,313.222,-97.946,174.054,32.788,156.026
C07886=1066.247,313.470,-97.979,174.057,32.792,156.027
C07887=1066.254,313.717,-98.011,174.060,32.796,156.027
C07888=1066.260,313.965,-98.044,174.063,32.800,156.028
C07889=1066.266,314.213,-98.077,174.066,32.805,156.029
C07890=1066.272,314.460,-98.110,174.070,32.810,156.030
C07891=1066.278,314.708,-98.142,174.073,32.814,156.031
C07892=1066.284,314.956,-98.176,174.076,32.819,156.032
C07893=1066.291,315.204,-98.209,174.079,32.823,156.033
C07894=1066.296,315.452,-98.242,174.082,32.828,156.034
C07895=1066.303,315.700,-98.275,174.086,32.832,156.034
C07896=1066.309,315.947,-98.308,174.089,32.837,156.035
C07897=1066.315,316.194,-98.342,174.092,32.841,156.036
C07898=1066.321,316.442,-98.374,174.095,32.846,156.037
C07899=1066.327,316.690,-98.408,174.098,32.851,156.038
C07900=1066.333,316.938,-98.440,174.102,32.855,156.039
C07901=1066.339,317.171,-98.472,174.105,32.859,156.040
C07902=1066.345,317.406,-98.504,174.108,32.864,156.041
C07903=1066.350,317.640,-98.535,174.111,32.868,156.041
C07904=1066.357,317.874,-98.567,174.114,32.872,156.042
C07905=1066.362,318.109,-98.598,174.117,32.877,156.043
C07906=1066.368,318.342,-98.629,174.120,32.881,156.044
C07907=1066.374,318.576,-98.661,174.123,32.886,156.045
C07908=1066.380,318.811,-98.693,174.126,32.890,156.046
C07909=1066.386,319.058,-98.726,174.128,32.894,156.046
C07910=1066.392,319.306,-98.759,174.132,32.899,156.047
C07911=1066.398,319.554,-98.792,174.135,32.904,156.048
C07912=1066.405,319.802,-98.826,174.138,32.908,156.049
C07913=1066.411,320.049,-98.859,174.141,32.913,156.050
C07914=1066.417,320.297,-98.893,174.145,32.917,156.051
C07915=1066.423,320.544,-98.926,174.148,32.922,156.052
C07916=1066.429,320.793,-98.960,174.151,32.926,156.053
C07917=1066.436,321.040,-98.993,174.154,32.931,156.054
C07918=1066.441,321.288,-99.027,174.158,32.935,156.054
C07919=1066.448,321.535,-99.060,174.161,32.940,156.055
C07920=1066.454,321.783,-99.094,174.164,32.945,156.056
C07921=1066.461,322.030,-99.127,174.168,32.949,156.057
C07922=1066.467,322.279,-99.161,174.171,32.954,156.058
C07923=1066.473,322.526,-99.194,174.174,32.959,156.059
C07924=1066.479,322.773,-99.228,174.177,32.963,156.060
C07925=1066.486,323.021,-99.261,174.181,32.968,156.061
C07926=1066.492,323.269,-99.296,174.185,32.972,156.062
C07927=1066.498,323.516,-99.328,174.188,32.977,156.063
C07928=1066.505,323.764,-99.363,174.192,32.982,156.064
C07929=1066.511,324.011,-99.396,174.195,32.986,156.064
C07930=1066.518,324.260,-99.430,174.198,32.991,156.065
C07931=1066.523,324.507,-99.464,174.202,32.996,156.066
C07932=1066.531,324.755,-99.498,174.205,33.000,156.067
C07933=1066.536,325.003,-99.531,174.208,33.005,156.068
C07934=1066.543,325.250,-99.565,174.212,33.009,156.069
C07935=1066.549,325.498,-99.599,174.215,33.014,156.070
C07936=1066.556,325.745,-99.632,174.218,33.019,156.071
C07937=1066.562,325.993,-99.667,174.222,33.024,156.072
C07938=1066.568,326.240,-99.700,174.225,33.028,156.073
C07939=1066.575,326.488,-99.734,174.228,33.033,156.074
C07940=1066.581,326.736,-99.768,174.232,33.037,156.075
C07941=1066.588,326.983,-99.802,174.235,33.042,156.075
C07942=1066.595,327.231,-99.836,174.238,33.047,156.076
C07943=1066.600,327.478,-99.870,174.242,33.052,156.077
C07944=1066.608,327.726,-99.904,174.245,33.056,156.078
C07945=1066.613,327.974,-99.938,174.249,33.061,156.079
C07946=1066.620,328.222,-99.971,174.252,33.065,156.080
C07947=1066.626,328.469,-100.005,174.255,33.070,156.081
C07948=1066.633,328.717,-100.040,174.259,33.075,156.082
C07949=1066.640,328.965,-100.074,174.262,33.080,156.083
C07950=1066.646,329.212,-100.108,174.266,33.085,156.084
C07951=1066.652,329.460,-100.142,174.269,33.089,156.085
C07952=1066.659,329.707,-100.176,174.272,33.094,156.086
C07953=1066.665,329.955,-100.210,174.276,33.099,156.087
C07954=1066.672,330.202,-100.245,174.279,33.103,156.088
C07955=1066.679,330.449,-100.279,174.283,33.108,156.089
C07956=1066.685,330.697,-100.313,174.286,33.113,156.089
C07957=1066.691,330.929,-100.344,174.289,33.117,156.090
C07958=1066.697,331.160,-100.377,174.292,33.122,156.091
C07959=1066.703,331.391,-100.409,174.296,33.126,156.092
C07960=1066.708,331.621,-100.441,174.299,33.131,156.093
C07961=1066.715,331.853,-100.473,174.302,33.136,156.094
C07962=1066.721,332.084,-100.505,174.305,33.140,156.095
C07963=1066.726,332.315,-100.538,174.308,33.144,156.096
C07964=1066.732,332.547,-100.570,174.312,33.149,156.097
C07965=1066.738,332.794,-100.604,174.315,33.154,156.098
C07966=1066.745,333.041,-100.639,174.318,33.159,156.099
C07967=1066.751,333.289,-100.674,174.323,33.164,156.100
C07968=1066.757,333.536,-100.708,174.326,33.169,156.101
C07969=1066.764,333.784,-100.743,174.330,33.173,156.102
C07970=1066.771,334.032,-100.777,174.333,33.178,156.102
C07971=1066.776,334.279,-100.811,174.337,33.184,156.104
C07972=1066.783,334.526,-100.847,174.340,33.188,156.104
C07973=1066.790,334.774,-100.881,174.344,33.193,156.105
C07974=1066.796,335.022,-100.916,174.347,33.198,156.106
C07975=1066.802,335.269,-100.950,174.351,33.203,156.107
C07976=1066.809,335.516,-100.985,174.354,33.208,156.108
C07977=1066.816,335.764,-101.020,174.358,33.213,156.109
C07978=1066.822,336.012,-101.055,174.361,33.218,156.110
C07979=1066.828,336.259,-101.089,174.365,33.223,156.111
C07980=1066.835,336.506,-101.124,174.368,33.228,156.112
C07981=1066.842,336.754,-101.159,174.371,33.232,156.113
C07982=1066.848,337.002,-101.194,174.375,33.238,156.114
C07983=1066.855,337.249,-101.229,174.379,33.243,156.115
C07984=1066.860,337.497,-101.263,174.382,33.248,156.116
C07985=1066.867,337.744,-101.299,174.385,33.253,156.117
C07986=1066.874,337.991,-101.334,174.390,33.258,156.118
C07987=1066.880,338.239,-101.368,174.394,33.263,156.119
C07988=1066.886,338.487,-101.404,174.397,33.268,156.121
C07989=1066.892,338.734,-101.439,174.401,33.273,156.121
C07990=1066.899,338.981,-101.474,174.404,33.278,156.123
C07991=1066.906,339.229,-101.509,174.408,33.283,156.124
C07992=1066.911,339.477,-101.544,174.411,33.288,156.125
C07993=1066.918,339.724,-101.579,174.415,33.293,156.126
C07994=1066.925,339.972,-101.614,174.418,33.298,156.127
C07995=1066.930,340.219,-101.649,174.422,33.303,156.128
C07996=1066.937,340.466,-101.685,174.425,33.308,156.129
C07997=1066.944,340.713,-101.720,174.429,33.313,156.130
C07998=1066.950,340.961,-101.755,174.432,33.318,156.131
C07999=1066.957,341.208,-101.791,174.436,33.324,156.132
C08000=1066.964,341.456,-101.826,174.440,33.329,156.133
C08001=1066.969,341.704,-101.861,174.444,33.334,156.134
C08002=1066.976,341.951,-101.896,174.448,33.339,156.135
C08003=1066.983,342.199,-101.931,174.451,33.344,156.136
C08004=1066.989,342.446,-101.967,174.455,33.349,156.137
C08005=1066.996,342.693,-102.003,174.458,33.354,156.138
C08006=1067.003,342.940,-102.038,174.462,33.360,156.139
C08007=1067.009,343.188,-102.073,174.465,33.365,156.140
C08008=1067.015,343.436,-102.109,174.469,33.370,156.141
C08009=1067.022,343.683,-102.144,174.473,33.375,156.142
C08010=1067.028,343.931,-102.179,174.476,33.380,156.143
C08011=1067.035,344.178,-102.215,174.481,33.385,156.144
C08012=1067.041,344.426,-102.250,174.484,33.391,156.145
C08013=1067.047,344.654,-102.283,174.488,33.395,156.146
C08014=1067.052,344.882,-102.316,174.491,33.401,156.147
C08015=1067.059,345.111,-102.349,174.494,33.405,156.148
C08016=1067.065,345.339,-102.382,174.498,33.410,156.149
C08017=1067.071,345.569,-102.415,174.501,33.415,156.150
C08018=1067.077,345.797,-102.448,174.504,33.420,156.151
C08019=1067.083,346.026,-102.482,174.508,33.425,156.152
C08020=1067.089,346.254,-102.514,174.511,33.430,156.153
C08021=1067.095,346.502,-102.550,174.515,33.435,156.155
C08022=1067.102,346.749,-102.586,174.519,33.440,156.156
C08023=1067.108,346.996,-102.622,174.523,33.446,156.157
C08024=1067.114,347.243,-102.658,174.527,33.451,156.158
C08025=1067.121,347.491,-102.693,174.530,33.456,156.159
C08026=1067.128,347.739,-102.729,174.534,33.461,156.160
C08027=1067.135,347.986,-102.765,174.538,33.467,156.161
C08028=1067.141,348.234,-102.801,174.541,33.472,156.162
C08029=1067.147,348.481,-102.837,174.545,33.478,156.163
C08030=1067.154,348.728,-102.874,174.549,33.483,156.164
C08031=1067.160,348.975,-102.909,174.553,33.488,156.165
C08032=1067.167,349.222,-102.945,174.557,33.494,156.167
C08033=1067.173,349.470,-102.981,174.561,33.499,156.168
C08034=1067.180,349.717,-103.017,174.564,33.504,156.169
C08035=1067.187,349.964,-103.054,174.568,33.510,156.170
C08036=1067.193,350.212,-103.089,174.572,33.516,156.171
C08037=1067.200,350.459,-103.125,174.575,33.521,156.172
C08038=1067.206,350.706,-103.162,174.579,33.526,156.173
C08039=1067.213,350.954,-103.198,174.584,33.532,156.174
C08040=1067.219,351.201,-103.234,174.588,33.537,156.176
C08041=1067.226,351.448,-103.270,174.591,33.542,156.177
C08042=1067.233,351.695,-103.307,174.595,33.548,156.178
C08043=1067.239,351.943,-103.343,174.599,33.553,156.179
C08044=1067.245,352.190,-103.379,174.602,33.559,156.180
C08045=1067.252,352.438,-103.415,174.606,33.564,156.181
C08046=1067.259,352.684,-103.451,174.611,33.570,156.182
C08047=1067.265,352.931,-103.488,174.615,33.575,156.183
C08048=1067.272,353.179,-103.525,174.618,33.581,156.185
C08049=1067.279,353.426,-103.561,174.622,33.586,156.186
C08050=1067.285,353.673,-103.597,174.626,33.592,156.187
C08051=1067.292,353.921,-103.634,174.630,33.598,156.188
C08052=1067.298,354.168,-103.671,174.633,33.603,156.189
C08053=1067.304,354.415,-103.707,174.638,33.609,156.190
C08054=1067.311,354.662,-103.744,174.642,33.615,156.192
C08055=1067.318,354.910,-103.780,174.646,33.620,156.193
C08056=1067.324,355.157,-103.817,174.649,33.626,156.194
C08057=1067.330,355.404,-103.853,174.653,33.632,156.195
C08058=1067.337,355.652,-103.890,174.657,33.637,156.196
C08059=1067.344,355.899,-103.927,174.661,33.643,156.197
C08060=1067.350,356.146,-103.963,174.665,33.648,156.199
C08061=1067.357,356.393,-104.001,174.669,33.654,156.200
C08062=1067.364,356.640,-104.037,174.673,33.660,156.201
C08063=1067.371,356.888,-104.074,174.677,33.666,156.202
C08064=1067.377,357.135,-104.110,174.681,33.671,156.203
C08065=1067.384,357.381,-104.147,174.684,33.677,156.205
C08066=1067.390,357.629,-104.184,174.689,33.682,156.206
C08067=1067.397,357.876,-104.221,174.693,33.688,156.207
C08068=1067.404,358.123,-104.258,174.697,33.694,156.208
C08069=1067.414,358.502,-104.314,174.703,33.703,156.210
C08070=1067.425,358.881,-104.371,174.710,33.711,156.212
C08071=1067.434,359.260,-104.427,174.716,33.721,156.214
C08072=1067.445,359.638,-104.485,174.721,33.729,156.216
C08073=1067.451,359.885,-104.521,174.725,33.735,156.217
C08074=1067.458,360.133,-104.559,174.729,33.741,156.218
C08075=1067.465,360.380,-104.595,174.734,33.747,156.219
C08076=1067.471,360.627,-104.633,174.738,33.753,156.221
C08077=1067.478,360.874,-104.670,174.742,33.759,156.222
C08078=1067.485,361.121,-104.707,174.746,33.764,156.223
C08079=1067.491,361.368,-104.744,174.749,33.770,156.224
C08080=1067.498,361.616,-104.782,174.754,33.776,156.226
C08081=1067.504,361.862,-104.819,174.758,33.782,156.227
C08082=1067.511,362.110,-104.856,174.762,33.788,156.228
C08083=1067.518,362.356,-104.893,174.766,33.794,156.229
C08084=1067.524,362.604,-104.931,174.770,33.800,156.231
C08085=1067.532,362.851,-104.969,174.775,33.806,156.232
C08086=1067.538,363.098,-105.005,174.779,33.811,156.233
C08087=1067.545,363.345,-105.043,174.783,33.818,156.234
C08088=1067.551,363.592,-105.080,174.786,33.823,156.236
C08089=1067.558,363.839,-105.118,174.791,33.830,156.237
C08090=1067.566,364.086,-105.156,174.795,33.835,156.238
C08091=1067.572,364.333,-105.193,174.799,33.842,156.239
C08092=1067.579,364.581,-105.230,174.803,33.847,156.241
C08093=1067.588,364.910,-105.280,174.808,33.855,156.242
C08094=1067.596,365.239,-105.331,174.815,33.864,156.244
C08095=1067.605,365.569,-105.381,174.820,33.872,156.246
C08096=1067.614,365.899,-105.432,174.825,33.880,156.248
C08097=1067.621,366.146,-105.469,174.830,33.886,156.249
C08098=1067.627,366.392,-105.507,174.834,33.893,156.250
C08099=1067.634,366.639,-105.545,174.838,33.898,156.252
C08100=1067.641,366.886,-105.583,174.842,33.905,156.253
C08101=1067.648,367.133,-105.620,174.847,33.911,156.254
C08102=1067.654,367.380,-105.659,174.851,33.917,156.256
C08103=1067.661,367.627,-105.696,174.855,33.923,156.257
C08104=1067.668,367.875,-105.734,174.859,33.929,156.258
C08105=1067.674,368.121,-105.773,174.864,33.935,156.260
C08106=1067.681,368.368,-105.810,174.868,33.942,156.261
C08107=1067.688,368.616,-105.848,174.872,33.948,156.262
C08108=1067.695,368.862,-105.887,174.876,33.954,156.264
C08109=1067.701,369.109,-105.924,174.881,33.961,156.265
C08110=1067.708,369.356,-105.962,174.885,33.967,156.266
C08111=1067.715,369.603,-106.001,174.889,33.973,156.268
C08112=1067.722,369.850,-106.039,174.893,33.979,156.269
C08113=1067.729,370.097,-106.076,174.898,33.986,156.270
C08114=1067.736,370.344,-106.115,174.902,33.992,156.272
C08115=1067.742,370.591,-106.152,174.906,33.998,156.273
C08116=1067.749,370.837,-106.191,174.911,34.004,156.274
C08117=1067.756,371.085,-106.229,174.915,34.011,156.276
C08118=1067.763,371.331,-106.268,174.919,34.017,156.277
C08119=1067.770,371.579,-106.306,174.923,34.024,156.279
C08120=1067.777,371.826,-106.344,174.928,34.030,156.280
C08121=1067.784,372.065,-106.381,174.932,34.036,156.281
C08122=1067.790,372.304,-106.419,174.936,34.042,156.283
C08123=1067.797,372.544,-106.456,174.940,34.049,156.284
C08124=1067.804,372.783,-106.493,174.945,34.055,156.285
C08125=1067.811,373.022,-106.530,174.949,34.061,156.287
C08126=1067.817,373.261,-106.567,174.953,34.067,156.288
C08127=1067.823,373.500,-106.605,174.958,34.074,156.289
C08128=1067.830,373.740,-106.642,174.962,34.080,156.291
C08129=1067.836,373.986,-106.681,174.966,34.087,156.292
C08130=1067.843,374.233,-106.719,174.971,34.093,156.294
C08131=1067.850,374.480,-106.758,174.975,34.100,156.295
C08132=1067.857,374.727,-106.797,174.979,34.106,156.297
C08133=1067.864,374.974,-106.836,174.983,34.113,156.298
C08134=1067.871,375.220,-106.874,174.988,34.119,156.299
C08135=1067.878,375.467,-106.913,174.992,34.126,156.301
C08136=1067.885,375.714,-106.952,174.996,34.133,156.302
C08137=1067.892,375.961,-106.991,175.002,34.139,156.304
C08138=1067.899,376.208,-107.030,175.006,34.146,156.305
C08139=1067.905,376.454,-107.068,175.010,34.153,156.307
C08140=1067.912,376.701,-107.107,175.015,34.160,156.308
C08141=1067.919,376.948,-107.146,175.019,34.166,156.310
C08142=1067.926,377.195,-107.185,175.023,34.173,156.311
C08143=1067.933,377.442,-107.224,175.028,34.179,156.312
C08144=1067.939,377.688,-107.263,175.033,34.186,156.314
C08145=1067.947,377.936,-107.302,175.037,34.193,156.315
C08146=1067.954,378.182,-107.341,175.042,34.200,156.317
C08147=1067.961,378.429,-107.380,175.046,34.206,156.318
C08148=1067.968,378.676,-107.419,175.051,34.213,156.320
C08149=1067.974,378.923,-107.458,175.055,34.220,156.321
C08150=1067.981,379.169,-107.497,175.060,34.227,156.323
C08151=1067.988,379.416,-107.536,175.065,34.234,156.324
C08152=1067.996,379.663,-107.575,175.069,34.241,156.326
C08153=1068.003,379.909,-107.615,175.073,34.247,156.327
C08154=1068.010,380.156,-107.654,175.079,34.254,156.329
C08155=1068.017,380.402,-107.693,175.083,34.261,156.330
C08156=1068.024,380.650,-107.733,175.087,34.268,156.332
C08157=1068.031,380.897,-107.771,175.092,34.275,156.334
C08158=1068.038,381.143,-107.811,175.096,34.282,156.335
C08159=1068.045,381.390,-107.850,175.102,34.289,156.337
C08160=1068.052,381.637,-107.890,175.106,34.296,156.338
C08161=1068.059,381.883,-107.930,175.110,34.303,156.340
C08162=1068.066,382.130,-107.969,175.115,34.310,156.341
C08163=1068.072,382.377,-108.009,175.120,34.317,156.343
C08164=1068.080,382.624,-108.048,175.125,34.324,156.344
C08165=1068.087,382.870,-108.088,175.129,34.331,156.346
C08166=1068.093,383.117,-108.128,175.133,34.338,156.348
C08167=1068.100,383.363,-108.167,175.139,34.345,156.349
C08168=1068.108,383.611,-108.207,175.143,34.352,156.351
C08169=1068.114,383.857,-108.247,175.148,34.360,156.352
C08170=1068.121,384.103,-108.286,175.153,34.367,156.354
C08171=1068.129,384.350,-108.326,175.158,34.374,156.356
C08172=1068.135,384.597,-108.366,175.162,34.381,156.357
C08173=1068.142,384.843,-108.406,175.166,34.388,156.359
C08174=1068.149,385.090,-108.446,175.172,34.395,156.360
C08175=1068.156,385.336,-108.486,175.176,34.403,156.362
C08176=1068.164,385.584,-108.525,175.181,34.410,156.364
C08177=1068.171,385.845,-108.568,175.186,34.418,156.365
C08178=1068.178,386.107,-108.610,175.192,34.425,156.367
C08179=1068.187,386.369,-108.653,175.196,34.433,156.369
C08180=1068.193,386.631,-108.695,175.202,34.441,156.371
C08181=1068.201,386.877,-108.735,175.206,34.448,156.372
C08182=1068.208,387.124,-108.775,175.211,34.456,156.374
C08183=1068.215,387.371,-108.815,175.216,34.463,156.375
C08184=1068.222,387.616,-108.856,175.220,34.470,156.377
C08185=1068.229,387.864,-108.896,175.226,34.478,156.379
C08186=1068.237,388.110,-108.936,175.230,34.485,156.380
C08187=1068.244,388.357,-108.976,175.236,34.492,156.382
C08188=1068.251,388.603,-109.016,175.240,34.500,156.384
C08189=1068.259,388.850,-109.056,175.245,34.507,156.385
C08190=1068.265,389.096,-109.096,175.250,34.515,156.387
C08191=1068.273,389.342,-109.137,175.255,34.522,156.389
C08192=1068.280,389.590,-109.178,175.260,34.530,156.390
C08193=1068.287,389.836,-109.217,175.265,34.537,156.392
C08194=1068.295,390.082,-109.258,175.270,34.545,156.394
C08195=1068.302,390.329,-109.298,175.275,34.552,156.396
C08196=1068.309,390.575,-109.339,175.280,34.560,156.397
C08197=1068.317,390.822,-109.379,175.285,34.567,156.399
C08198=1068.323,391.068,-109.420,175.289,34.575,156.401
C08199=1068.330,391.315,-109.460,175.295,34.583,156.402
C08200=1068.338,391.561,-109.501,175.299,34.591,156.404
C08201=1068.345,391.807,-109.542,175.305,34.598,156.406
C08202=1068.352,392.055,-109.582,175.309,34.605,156.408
C08203=1068.360,392.301,-109.623,175.315,34.613,156.409
C08204=1068.367,392.547,-109.664,175.319,34.621,156.411
C08205=1068.374,392.794,-109.704,175.325,34.629,156.413
C08206=1068.381,393.041,-109.746,175.330,34.637,156.415
C08207=1068.388,393.286,-109.786,175.335,34.645,156.417
C08208=1068.396,393.533,-109.827,175.340,34.652,156.418
C08209=1068.403,393.779,-109.868,175.345,34.660,156.420
C08210=1068.410,394.027,-109.909,175.350,34.668,156.422
C08211=1068.417,394.273,-109.950,175.355,34.676,156.424
C08212=1068.425,394.519,-109.990,175.360,34.684,156.426
C08213=1068.432,394.765,-110.032,175.365,34.692,156.427
C08214=1068.439,395.012,-110.073,175.371,34.700,156.429
C08215=1068.447,395.259,-110.114,175.376,34.708,156.431
C08216=1068.454,395.505,-110.155,175.381,34.716,156.433
C08217=1068.461,395.751,-110.196,175.386,34.724,156.435
C08218=1068.468,395.998,-110.237,175.391,34.732,156.437
C08219=1068.475,396.244,-110.279,175.396,34.740,156.438
C08220=1068.483,396.490,-110.321,175.402,34.748,156.440
C08221=1068.490,396.737,-110.362,175.407,34.756,156.442
C08222=1068.497,396.983,-110.403,175.412,34.764,156.444
C08223=1068.505,397.230,-110.444,175.417,34.772,156.446
C08224=1068.513,397.476,-110.485,175.422,34.780,156.448
C08225=1068.520,397.722,-110.527,175.428,34.789,156.450
C08226=1068.527,397.969,-110.568,175.433,34.797,156.451
C08227=1068.535,398.215,-110.609,175.438,34.805,156.453
C08228=1068.542,398.462,-110.652,175.444,34.813,156.455
C08229=1068.549,398.708,-110.693,175.449,34.822,156.457
C08230=1068.556,398.954,-110.735,175.454,34.830,156.459
C08231=1068.564,399.201,-110.776,175.460,34.838,156.461
C08232=1068.571,399.447,-110.818,175.464,34.846,156.463
C08233=1068.579,399.725,-110.865,175.471,34.856,156.465
C08234=1068.588,400.003,-110.912,175.477,34.865,156.467
C08235=1068.596,400.281,-110.959,175.483,34.875,156.469
C08236=1068.605,400.558,-111.006,175.489,34.884,156.472
C08237=1068.612,400.804,-111.048,175.494,34.893,156.474
C08238=1068.619,401.051,-111.090,175.500,34.901,156.476
C08239=1068.626,401.297,-111.132,175.505,34.910,156.478
C08240=1068.635,401.544,-111.174,175.510,34.918,156.480
C08241=1068.642,401.790,-111.216,175.516,34.927,156.482
C08242=1068.650,402.037,-111.257,175.522,34.935,156.483
C08243=1068.656,402.283,-111.300,175.527,34.944,156.485
C08244=1068.664,402.529,-111.342,175.532,34.952,156.488
C08245=1068.672,402.775,-111.384,175.538,34.961,156.489
C08246=1068.680,403.021,-111.426,175.543,34.969,156.491
C08247=1068.687,403.268,-111.468,175.549,34.978,156.494
C08248=1068.694,403.514,-111.510,175.554,34.987,156.496
C08249=1068.702,403.761,-111.552,175.560,34.995,156.498
C08250=1068.709,404.007,-111.594,175.565,35.004,156.500
C08251=1068.717,404.253,-111.636,175.571,35.013,156.502
C08252=1068.725,404.499,-111.679,175.577,35.022,156.504
C08253=1068.732,404.746,-111.722,175.582,35.031,156.506
C08254=1068.739,404.992,-111.764,175.587,35.039,156.508
C08255=1068.747,405.239,-111.807,175.593,35.048,156.510
C08256=1068.755,405.485,-111.849,175.599,35.057,156.512
C08257=1068.761,405.731,-111.891,175.605,35.066,156.514
C08258=1068.770,405.977,-111.934,175.611,35.075,156.516
C08259=1068.777,406.223,-111.977,175.616,35.084,156.518
C08260=1068.785,406.470,-112.019,175.621,35.093,156.521
C08261=1068.792,406.716,-112.062,175.627,35.102,156.523
C08262=1068.800,406.962,-112.105,175.633,35.111,156.525
C08263=1068.807,407.208,-112.147,175.639,35.120,156.527
C08264=1068.814,407.454,-112.191,175.645,35.129,156.529
C08265=1068.823,407.701,-112.233,175.650,35.138,156.531
C08266=1068.830,407.946,-112.276,175.656,35.148,156.533
C08267=1068.837,408.193,-112.319,175.662,35.157,156.536
C08268=1068.845,408.439,-112.362,175.668,35.166,156.538
C08269=1068.853,408.686,-112.405,175.674,35.175,156.540
C08270=1068.860,408.931,-112.448,175.680,35.184,156.542
C08271=1068.868,409.178,-112.491,175.686,35.194,156.544
C08272=1068.876,409.425,-112.534,175.691,35.203,156.547
C08273=1068.883,409.670,-112.577,175.697,35.212,156.549
C08274=1068.891,409.916,-112.620,175.703,35.222,156.551
C08275=1068.898,410.162,-112.663,175.709,35.231,156.553
C08276=1068.906,410.409,-112.706,175.715,35.240,156.555
C08277=1068.914,410.655,-112.749,175.721,35.250,156.558
C08278=1068.922,410.901,-112.793,175.727,35.259,156.560
C08279=1068.929,411.147,-112.836,175.733,35.269,156.562
C08280=1068.937,411.393,-112.880,175.739,35.278,156.564
C08281=1068.945,411.639,-112.922,175.745,35.288,156.567
C08282=1068.953,411.885,-112.966,175.751,35.297,156.569
C08283=1068.961,412.131,-113.010,175.757,35.306,156.571
C08284=1068.968,412.378,-113.053,175.763,35.316,156.574
C08285=1068.976,412.623,-113.096,175.769,35.326,156.576
C08286=1068.984,412.869,-113.140,175.776,35.335,156.578
C08287=1068.992,413.116,-113.183,175.781,35.345,156.581
C08288=1068.999,413.362,-113.227,175.787,35.355,156.583
C08289=1069.008,413.644,-113.277,175.795,35.366,156.586
C08290=1069.018,413.926,-113.327,175.802,35.377,156.588
C08291=1069.027,414.208,-113.377,175.809,35.388,156.591
C08292=1069.036,414.489,-113.427,175.816,35.399,156.594
C08293=1069.044,414.735,-113.470,175.822,35.409,156.596
C08294=1069.052,414.981,-113.514,175.828,35.419,156.598
C08295=1069.060,415.227,-113.558,175.834,35.429,156.601
C08296=1069.067,415.473,-113.603,175.840,35.439,156.603
C08297=1069.075,415.720,-113.646,175.847,35.449,156.606
C08298=1069.083,415.965,-113.691,175.853,35.459,156.608
C08299=1069.091,416.211,-113.735,175.859,35.469,156.611
C08300=1069.099,416.458,-113.779,175.866,35.479,156.613
C08301=1069.107,416.703,-113.823,175.873,35.489,156.615
C08302=1069.115,416.949,-113.867,175.879,35.499,156.618
C08303=1069.123,417.195,-113.911,175.885,35.509,156.620
C08304=1069.131,417.441,-113.955,175.892,35.519,156.623
C08305=1069.139,417.687,-114.000,175.898,35.530,156.625
C08306=1069.147,417.933,-114.044,175.904,35.540,156.628
C08307=1069.154,418.179,-114.089,175.911,35.550,156.630
C08308=1069.162,418.424,-114.133,175.917,35.561,156.633
C08309=1069.170,418.671,-114.177,175.924,35.571,156.635
C08310=1069.178,418.917,-114.221,175.931,35.581,156.638
C08311=1069.186,419.162,-114.265,175.937,35.592,156.640
C08312=1069.194,419.408,-114.310,175.943,35.602,156.643
C08313=1069.203,419.654,-114.355,175.950,35.612,156.645
C08314=1069.211,419.900,-114.400,175.956,35.623,156.648
C08315=1069.219,420.146,-114.444,175.964,35.634,156.651
C08316=1069.227,420.391,-114.489,175.970,35.644,156.653
C08317=1069.235,420.637,-114.533,175.977,35.654,156.656
C08318=1069.244,420.884,-114.578,175.983,35.665,156.658
C08319=1069.251,421.129,-114.623,175.991,35.676,156.661
C08320=1069.259,421.375,-114.668,175.997,35.686,156.664
C08321=1069.268,421.621,-114.712,176.004,35.697,156.666
C08322=1069.276,421.867,-114.758,176.010,35.708,156.669
C08323=1069.284,422.112,-114.802,176.018,35.719,156.672
C08324=1069.291,422.358,-114.848,176.024,35.729,156.674
C08325=1069.300,422.604,-114.893,176.031,35.740,156.677
C08326=1069.308,422.850,-114.938,176.037,35.751,156.680
C08327=1069.316,423.095,-114.983,176.045,35.762,156.682
C08328=1069.325,423.341,-115.028,176.051,35.773,156.685
C08329=1069.332,423.587,-115.074,176.058,35.784,156.688
C08330=1069.340,423.832,-115.118,176.066,35.795,156.690
C08331=1069.349,424.079,-115.164,176.072,35.806,156.693
C08332=1069.357,424.324,-115.209,176.079,35.817,156.696
C08333=1069.365,424.570,-115.255,176.086,35.828,156.699
C08334=1069.374,424.815,-115.300,176.093,35.840,156.702
C08335=1069.382,425.062,-115.346,176.101,35.851,156.704
C08336=1069.390,425.307,-115.391,176.107,35.862,156.707
C08337=1069.398,425.553,-115.437,176.114,35.873,156.710
C08338=1069.407,425.798,-115.482,176.122,35.884,156.713
C08339=1069.415,426.044,-115.528,176.129,35.896,156.715
C08340=1069.423,426.289,-115.573,176.136,35.907,156.718
C08341=1069.431,426.536,-115.619,176.143,35.918,156.721
C08342=1069.441,426.781,-115.665,176.151,35.929,156.724
C08343=1069.448,427.026,-115.711,176.158,35.941,156.727
C08344=1069.457,427.272,-115.756,176.165,35.952,156.730
C08345=1069.468,427.573,-115.813,176.173,35.966,156.733
C08346=1069.478,427.874,-115.869,176.182,35.980,156.737
C08347=1069.488,428.175,-115.925,176.192,35.995,156.740
C08348=1069.498,428.475,-115.982,176.201,36.009,156.744
C08349=1069.506,428.721,-116.028,176.208,36.021,156.747
C08350=1069.515,428.966,-116.074,176.215,36.032,156.750
C08351=1069.523,429.213,-116.120,176.223,36.044,156.753
C08352=1069.532,429.458,-116.166,176.230,36.056,156.756
C08353=1069.540,429.703,-116.212,176.238,36.068,156.759
C08354=1069.548,429.949,-116.259,176.245,36.080,156.762
C08355=1069.557,430.194,-116.306,176.253,36.092,156.765
C08356=1069.565,430.440,-116.352,176.261,36.103,156.768
C08357=1069.574,430.686,-116.398,176.268,36.115,156.771
C08358=1069.583,430.931,-116.444,176.276,36.127,156.774
C08359=1069.591,431.176,-116.491,176.283,36.139,156.777
C08360=1069.599,431.421,-116.537,176.291,36.151,156.780
C08361=1069.608,431.667,-116.584,176.299,36.163,156.783
C08362=1069.616,431.912,-116.631,176.307,36.176,156.786
C08363=1069.625,432.158,-116.678,176.314,36.188,156.789
C08364=1069.634,432.403,-116.724,176.322,36.201,156.792
C08365=1069.642,432.649,-116.771,176.330,36.213,156.796
C08366=1069.651,432.894,-116.818,176.337,36.225,156.799
C08367=1069.659,433.139,-116.865,176.345,36.238,156.802
C08368=1069.668,433.385,-116.912,176.353,36.250,156.805
C08369=1069.677,433.630,-116.959,176.361,36.262,156.808
C08370=1069.685,433.875,-117.006,176.369,36.275,156.811
C08371=1069.694,434.121,-117.053,176.376,36.287,156.815
C08372=1069.703,434.366,-117.100,176.385,36.300,156.818
C08373=1069.711,434.612,-117.148,176.393,36.313,156.821
C08374=1069.719,434.857,-117.194,176.401,36.325,156.824
C08375=1069.728,435.102,-117.242,176.409,36.338,156.828
C08376=1069.737,435.347,-117.289,176.417,36.351,156.831
C08377=1069.746,435.593,-117.336,176.425,36.363,156.834
C08378=1069.755,435.838,-117.384,176.433,36.376,156.838
C08379=1069.764,436.083,-117.431,176.441,36.389,156.841
C08380=1069.772,436.328,-117.478,176.449,36.402,156.844
C08381=1069.781,436.574,-117.526,176.458,36.415,156.848
C08382=1069.790,436.819,-117.574,176.466,36.428,156.851
C08383=1069.799,437.064,-117.621,176.474,36.441,156.854
C08384=1069.808,437.309,-117.669,176.483,36.454,156.858
C08385=1069.817,437.554,-117.717,176.491,36.467,156.861
C08386=1069.826,437.799,-117.764,176.499,36.480,156.864
C08387=1069.835,438.045,-117.812,176.508,36.493,156.868
C08388=1069.843,438.290,-117.860,176.516,36.506,156.871
C08389=1069.852,438.535,-117.907,176.525,36.519,156.875
C08390=1069.862,438.781,-117.955,176.533,36.533,156.878
C08391=1069.870,439.025,-118.004,176.541,36.546,156.882
C08392=1069.880,439.271,-118.052,176.550,36.559,156.885
C08393=1069.888,439.516,-118.099,176.559,36.573,156.889
C08394=1069.897,439.761,-118.148,176.568,36.587,156.892
C08395=1069.906,440.006,-118.196,176.576,36.600,156.896
C08396=1069.915,440.251,-118.245,176.585,36.613,156.899
C08397=1069.924,440.496,-118.292,176.593,36.627,156.903
C08398=1069.934,440.741,-118.341,176.602,36.641,156.907
C08399=1069.942,440.986,-118.389,176.611,36.655,156.910
C08400=1069.952,441.231,-118.437,176.620,36.668,156.914
C08401=1069.959,441.446,-118.480,176.628,36.680,156.917
C08402=1069.967,441.661,-118.522,176.636,36.693,156.920
C08403=1069.975,441.875,-118.565,176.643,36.705,156.923
C08404=1069.984,442.090,-118.608,176.651,36.717,156.927
C08405=1069.992,442.305,-118.650,176.659,36.729,156.930
C08406=1069.999,442.520,-118.693,176.667,36.741,156.933
C08407=1070.007,442.734,-118.736,176.675,36.754,156.936
C08408=1070.016,442.949,-118.779,176.683,36.766,156.940
C08409=1070.024,443.193,-118.827,176.691,36.780,156.943
C08410=1070.034,443.438,-118.876,176.701,36.794,156.947
C08411=1070.043,443.684,-118.925,176.710,36.808,156.951
C08412=1070.052,443.929,-118.974,176.720,36.823,156.955
C08413=1070.062,444.173,-119.023,176.728,36.837,156.959
C08414=1070.071,444.418,-119.072,176.738,36.851,156.962
C08415=1070.080,444.663,-119.121,176.747,36.866,156.966
C08416=1070.090,444.908,-119.170,176.757,36.881,156.970
C08417=1070.099,445.153,-119.220,176.766,36.895,156.974
C08418=1070.108,445.397,-119.269,176.776,36.910,156.978
C08419=1070.117,445.643,-119.319,176.784,36.924,156.982
C08420=1070.127,445.887,-119.368,176.794,36.939,156.986
C08421=1070.136,446.132,-119.418,176.803,36.954,156.990
C08422=1070.145,446.377,-119.467,176.813,36.968,156.994
C08423=1070.155,446.622,-119.517,176.823,36.983,156.998
C08424=1070.164,446.866,-119.566,176.832,36.998,157.002
C08425=1070.174,447.111,-119.616,176.842,37.013,157.006
C08426=1070.183,447.355,-119.665,176.852,37.028,157.010
C08427=1070.192,447.601,-119.715,176.861,37.043,157.014
C08428=1070.202,447.846,-119.765,176.871,37.058,157.018
C08429=1070.212,448.089,-119.814,176.881,37.073,157.022
C08430=1070.222,448.332,-119.864,176.891,37.088,157.026
C08431=1070.233,448.577,-119.913,176.899,37.102,157.030
C08432=1070.245,448.822,-119.961,176.908,37.117,157.034
C08433=1070.259,449.066,-120.008,176.916,37.130,157.037
C08434=1070.273,449.311,-120.055,176.925,37.143,157.041
C08435=1070.289,449.556,-120.101,176.933,37.156,157.044
C08436=1070.306,449.802,-120.146,176.940,37.168,157.048
C08437=1069.957,449.802,-120.399,176.927,37.307,157.085
C08438=1069.941,449.557,-120.354,176.920,37.295,157.081
C08439=1069.925,449.312,-120.308,176.911,37.282,157.078
C08440=1069.911,449.067,-120.261,176.903,37.269,157.074
C08441=1069.897,448.822,-120.214,176.894,37.255,157.071
C08442=1069.885,448.577,-120.165,176.886,37.241,157.067
C08443=1069.873,448.332,-120.116,176.876,37.227,157.063
C08444=1069.863,448.088,-120.068,176.866,37.212,157.059
C08445=1069.853,447.845,-120.018,176.856,37.197,157.055
C08446=1069.843,447.601,-119.968,176.847,37.182,157.051
C08447=1069.834,447.356,-119.918,176.837,37.167,157.047
C08448=1069.825,447.111,-119.869,176.827,37.152,157.043
C08449=1069.815,446.867,-119.819,176.817,37.137,157.039
C08450=1069.806,446.622,-119.769,176.807,37.122,157.035
C08451=1069.795,446.377,-119.719,176.798,37.108,157.031
C08452=1069.786,446.132,-119.670,176.788,37.093,157.027
C08453=1069.777,445.887,-119.620,176.778,37.078,157.023
C08454=1069.768,445.642,-119.571,176.769,37.063,157.019
C08455=1069.758,445.398,-119.521,176.759,37.049,157.015
C08456=1069.749,445.153,-119.472,176.749,37.034,157.011
C08457=1069.739,444.908,-119.422,176.741,37.020,157.007
C08458=1069.730,444.663,-119.373,176.731,37.005,157.003
C08459=1069.721,444.419,-119.324,176.722,36.991,156.999
C08460=1069.712,444.174,-119.275,176.712,36.977,156.995
C08461=1069.703,443.929,-119.225,176.703,36.962,156.991
C08462=1069.693,443.684,-119.177,176.693,36.948,156.988
C08463=1069.684,443.439,-119.128,176.685,36.934,156.984
C08464=1069.675,443.194,-119.079,176.675,36.920,156.980
C08465=1069.665,442.949,-119.030,176.666,36.905,156.976
C08466=1069.650,442.539,-118.948,176.651,36.882,156.970
C08467=1069.634,442.127,-118.867,176.636,36.859,156.964
C08468=1069.619,441.717,-118.785,176.621,36.835,156.958
C08469=1069.603,441.307,-118.704,176.606,36.812,156.952
C08470=1069.594,441.062,-118.655,176.596,36.798,156.948
C08471=1069.585,440.817,-118.607,176.587,36.785,156.944
C08472=1069.577,440.572,-118.558,176.579,36.771,156.941
C08473=1069.567,440.327,-118.510,176.569,36.758,156.937
C08474=1069.558,440.082,-118.461,176.561,36.744,156.933
C08475=1069.549,439.836,-118.413,176.552,36.730,156.930
C08476=1069.541,439.592,-118.364,176.544,36.717,156.926
C08477=1069.531,439.346,-118.317,176.535,36.704,156.923
C08478=1069.522,439.101,-118.269,176.526,36.690,156.919
C08479=1069.513,438.856,-118.220,176.517,36.677,156.916
C08480=1069.504,438.611,-118.173,176.509,36.663,156.912
C08481=1069.496,438.366,-118.125,176.500,36.650,156.909
C08482=1069.486,438.121,-118.076,176.492,36.637,156.905
C08483=1069.478,437.876,-118.029,176.484,36.624,156.902
C08484=1069.468,437.630,-117.981,176.475,36.611,156.899
C08485=1069.459,437.386,-117.933,176.467,36.598,156.895
C08486=1069.450,437.140,-117.886,176.457,36.585,156.892
C08487=1069.441,436.895,-117.838,176.449,36.572,156.888
C08488=1069.433,436.650,-117.790,176.441,36.559,156.885
C08489=1069.423,436.404,-117.742,176.433,36.546,156.882
C08490=1069.415,436.159,-117.696,176.424,36.533,156.878
C08491=1069.406,435.914,-117.648,176.416,36.520,156.875
C08492=1069.397,435.669,-117.601,176.408,36.508,156.872
C08493=1069.388,435.423,-117.553,176.399,36.495,156.868
C08494=1069.379,435.178,-117.506,176.391,36.482,156.865
C08495=1069.370,434.933,-117.459,176.384,36.469,156.862
C08496=1069.362,434.688,-117.411,176.376,36.457,156.858
C08497=1069.354,434.442,-117.364,176.368,36.444,156.855
C08498=1069.345,434.197,-117.316,176.359,36.432,156.852
C08499=1069.336,433.951,-117.269,176.351,36.419,156.849
C08500=1069.327,433.706,-117.222,176.343,36.407,156.846
C08501=1069.318,433.461,-117.175,176.335,36.394,156.842
C08502=1069.310,433.215,-117.128,176.327,36.382,156.839
C08503=1069.301,432.970,-117.081,176.319,36.369,156.836
C08504=1069.292,432.725,-117.034,176.312,36.357,156.833
C08505=1069.284,432.479,-116.988,176.304,36.345,156.830
C08506=1069.275,432.234,-116.941,176.296,36.332,156.826
C08507=1069.267,431.988,-116.894,176.288,36.320,156.823
C08508=1069.258,431.743,-116.847,176.281,36.308,156.820
C08509=1069.250,431.499,-116.800,176.273,36.296,156.817
C08510=1069.241,431.253,-116.754,176.265,36.284,156.814
C08511=1069.233,431.007,-116.708,176.257,36.272,156.811
C08512=1069.225,430.761,-116.661,176.250,36.260,156.808
C08513=1069.216,430.516,-116.614,176.242,36.248,156.805
C08514=1069.208,430.270,-116.567,176.234,36.236,156.802
C08515=1069.198,430.025,-116.521,176.227,36.224,156.799
C08516=1069.190,429.779,-116.475,176.219,36.212,156.796
C08517=1069.181,429.534,-116.428,176.211,36.200,156.793
C08518=1069.173,429.289,-116.382,176.204,36.188,156.790
C08519=1069.165,429.043,-116.337,176.196,36.177,156.787
C08520=1069.156,428.797,-116.290,176.188,36.165,156.784
C08521=1069.147,428.552,-116.243,176.182,36.154,156.781
C08522=1069.138,428.250,-116.186,176.172,36.139,156.777
C08523=1069.126,427.947,-116.130,176.163,36.125,156.774
C08524=1069.117,427.644,-116.074,176.154,36.111,156.770
C08525=1069.107,427.341,-116.017,176.145,36.096,156.767
C08526=1069.098,427.096,-115.971,176.137,36.085,156.764
C08527=1069.089,426.850,-115.924,176.130,36.074,156.761
C08528=1069.081,426.605,-115.879,176.123,36.062,156.758
C08529=1069.073,426.359,-115.833,176.116,36.051,156.755
C08530=1069.064,426.113,-115.788,176.108,36.040,156.752
C08531=1069.056,425.868,-115.742,176.101,36.028,156.749
C08532=1069.047,425.622,-115.697,176.094,36.017,156.747
C08533=1069.039,425.376,-115.651,176.087,36.006,156.744
C08534=1069.030,425.130,-115.606,176.079,35.995,156.741
C08535=1069.023,424.885,-115.560,176.073,35.984,156.738
C08536=1069.014,424.639,-115.515,176.066,35.973,156.735
C08537=1069.006,424.394,-115.469,176.058,35.961,156.733
C08538=1068.997,424.148,-115.424,176.052,35.950,156.730
C08539=1068.990,423.903,-115.378,176.044,35.939,156.727
C08540=1068.981,423.656,-115.333,176.037,35.928,156.724
C08541=1068.973,423.411,-115.288,176.030,35.918,156.722
C08542=1068.964,423.165,-115.242,176.023,35.906,156.719
C08543=1068.957,422.919,-115.197,176.017,35.896,156.716
C08544=1068.949,422.674,-115.152,176.009,35.885,156.714
C08545=1068.940,422.427,-115.106,176.003,35.874,156.711
C08546=1068.932,422.182,-115.062,175.996,35.863,156.708
C08547=1068.924,421.937,-115.017,175.989,35.852,156.706
C08548=1068.916,421.690,-114.972,175.982,35.842,156.703
C08549=1068.908,421.445,-114.927,175.975,35.831,156.700
C08550=1068.900,421.199,-114.882,175.968,35.820,156.698
C08551=1068.892,420.954,-114.837,175.962,35.809,156.695
C08552=1068.883,420.707,-114.792,175.955,35.799,156.692
C08553=1068.875,420.461,-114.748,175.948,35.789,156.690
C08554=1068.868,420.215,-114.703,175.941,35.778,156.687
C08555=1068.859,419.969,-114.658,175.935,35.767,156.685
C08556=1068.851,419.724,-114.613,175.928,35.757,156.682
C08557=1068.843,419.478,-114.569,175.921,35.747,156.679
C08558=1068.835,419.232,-114.524,175.914,35.736,156.677
C08559=1068.827,418.987,-114.480,175.908,35.726,156.674
C08560=1068.819,418.740,-114.435,175.902,35.716,156.672
C08561=1068.811,418.494,-114.390,175.895,35.705,156.669
C08562=1068.803,418.248,-114.346,175.888,35.695,156.667
C08563=1068.794,418.003,-114.302,175.882,35.685,156.664
C08564=1068.786,417.757,-114.257,175.875,35.675,156.662
C08565=1068.778,417.511,-114.213,175.869,35.664,156.659
C08566=1068.771,417.265,-114.169,175.863,35.654,156.657
C08567=1068.762,417.019,-114.125,175.855,35.644,156.654
C08568=1068.755,416.773,-114.080,175.849,35.634,156.652
C08569=1068.747,416.527,-114.036,175.843,35.624,156.649
C08570=1068.739,416.281,-113.992,175.836,35.614,156.647
C08571=1068.731,416.035,-113.948,175.830,35.604,156.644
C08572=1068.723,415.789,-113.903,175.824,35.593,156.642
C08573=1068.715,415.543,-113.860,175.818,35.584,156.640
C08574=1068.707,415.297,-113.815,175.811,35.574,156.637
C08575=1068.700,415.051,-113.772,175.804,35.564,156.635
C08576=1068.692,414.805,-113.727,175.798,35.554,156.632
C08577=1068.684,414.559,-113.684,175.792,35.544,156.630
C08578=1068.675,414.276,-113.634,175.785,35.533,156.627
C08579=1068.665,413.992,-113.583,175.778,35.522,156.625
C08580=1068.656,413.708,-113.533,175.771,35.510,156.622
C08581=1068.647,413.425,-113.482,175.763,35.499,156.619
C08582=1068.639,413.179,-113.439,175.757,35.489,156.617
C08583=1068.631,412.934,-113.395,175.751,35.480,156.614
C08584=1068.623,412.687,-113.351,175.745,35.470,156.612
C08585=1068.616,412.441,-113.308,175.738,35.461,156.610
C08586=1068.607,412.195,-113.265,175.732,35.451,156.608
C08587=1068.600,411.949,-113.222,175.726,35.441,156.605
C08588=1068.592,411.703,-113.178,175.720,35.432,156.603
C08589=1068.584,411.456,-113.134,175.714,35.423,156.601
C08590=1068.576,411.210,-113.091,175.708,35.413,156.598
C08591=1068.569,410.965,-113.048,175.702,35.404,156.596
C08592=1068.561,410.718,-113.004,175.696,35.394,156.594
C08593=1068.553,410.472,-112.961,175.690,35.385,156.592
C08594=1068.545,410.227,-112.918,175.684,35.375,156.589
C08595=1068.538,409.980,-112.875,175.678,35.366,156.587
C08596=1068.530,409.733,-112.832,175.672,35.357,156.585
C08597=1068.522,409.488,-112.789,175.667,35.348,156.583
C08598=1068.515,409.242,-112.745,175.661,35.338,156.580
C08599=1068.507,408.995,-112.702,175.655,35.329,156.578
C08600=1068.499,408.749,-112.660,175.649,35.320,156.576
C08601=1068.491,408.503,-112.616,175.643,35.310,156.574
C08602=1068.485,408.257,-112.574,175.637,35.301,156.572
C08603=1068.476,408.011,-112.531,175.631,35.292,156.569
C08604=1068.469,407.765,-112.487,175.625,35.283,156.567
C08605=1068.461,407.518,-112.444,175.619,35.274,156.565
C08606=1068.454,407.273,-112.402,175.613,35.265,156.563
C08607=1068.446,407.026,-112.359,175.607,35.256,156.561
C08608=1068.438,406.780,-112.316,175.602,35.246,156.559
C08609=1068.431,406.533,-112.273,175.597,35.238,156.557
C08610=1068.424,406.287,-112.231,175.591,35.229,156.554
C08611=1068.416,406.042,-112.188,175.585,35.220,156.552
C08612=1068.408,405.795,-112.145,175.579,35.211,156.550
C08613=1068.401,405.549,-112.103,175.573,35.202,156.548
C08614=1068.393,405.302,-112.060,175.567,35.193,156.546
C08615=1068.386,405.056,-112.018,175.562,35.184,156.544
C08616=1068.378,404.810,-111.976,175.557,35.175,156.542
C08617=1068.370,404.563,-111.933,175.551,35.167,156.540
C08618=1068.363,404.317,-111.891,175.545,35.158,156.538
C08619=1068.355,404.070,-111.848,175.539,35.149,156.536
C08620=1068.348,403.824,-111.806,175.533,35.140,156.533
C08621=1068.340,403.578,-111.764,175.529,35.131,156.531
C08622=1068.333,403.332,-111.722,175.523,35.123,156.529
C08623=1068.325,403.085,-111.679,175.517,35.114,156.527
C08624=1068.318,402.839,-111.637,175.511,35.106,156.525
C08625=1068.311,402.593,-111.595,175.506,35.097,156.523
C08626=1068.303,402.346,-111.552,175.501,35.088,156.521
C08627=1068.295,402.101,-111.510,175.495,35.080,156.519
C08628=1068.288,401.854,-111.469,175.489,35.071,156.517
C08629=1068.280,401.608,-111.427,175.484,35.063,156.515
C08630=1068.273,401.362,-111.385,175.479,35.054,156.513
C08631=1068.265,401.115,-111.342,175.473,35.046,156.511
C08632=1068.258,400.868,-111.301,175.467,35.037,156.509
C08633=1068.250,400.622,-111.259,175.463,35.029,156.507
C08634=1068.242,400.343,-111.212,175.456,35.019,156.505
C08635=1068.234,400.063,-111.164,175.450,35.010,156.503
C08636=1068.225,399.784,-111.116,175.444,35.000,156.501
C08637=1068.217,399.505,-111.069,175.437,34.991,156.499
C08638=1068.209,399.258,-111.028,175.433,34.983,156.497
C08639=1068.202,399.012,-110.986,175.427,34.974,156.495
C08640=1068.194,398.766,-110.945,175.421,34.966,156.493
C08641=1068.188,398.520,-110.902,175.416,34.958,156.491
C08642=1068.180,398.273,-110.861,175.411,34.949,156.489
C08643=1068.173,398.026,-110.820,175.406,34.941,156.487
C08644=1068.165,397.780,-110.778,175.400,34.933,156.485
C08645=1068.158,397.533,-110.736,175.395,34.925,156.483
C08646=1068.150,397.287,-110.695,175.390,34.917,156.481
C08647=1068.143,397.041,-110.653,175.384,34.909,156.480
C08648=1068.136,396.795,-110.612,175.380,34.900,156.478
C08649=1068.128,396.548,-110.572,175.374,34.893,156.476
C08650=1068.121,396.302,-110.531,175.368,34.884,156.474
C08651=1068.113,396.055,-110.489,175.364,34.876,156.472
C08652=1068.106,395.809,-110.447,175.358,34.869,156.470
C08653=1068.099,395.563,-110.406,175.353,34.860,156.468
C08654=1068.091,395.316,-110.365,175.348,34.853,156.467
C08655=1068.084,395.069,-110.324,175.343,34.844,156.465
C08656=1068.077,394.823,-110.282,175.338,34.837,156.463
C08657=1068.070,394.577,-110.242,175.332,34.829,156.461
C08658=1068.063,394.330,-110.200,175.327,34.821,156.459
C08659=1068.055,394.084,-110.159,175.322,34.813,156.457
C08660=1068.047,393.837,-110.119,175.317,34.805,156.456
C08661=1068.040,393.591,-110.077,175.312,34.797,156.454
C08662=1068.034,393.344,-110.037,175.307,34.789,156.452
C08663=1068.026,393.098,-109.996,175.301,34.781,156.450
C08664=1068.018,392.851,-109.955,175.297,34.774,156.448
C08665=1068.011,392.605,-109.914,175.291,34.766,156.447
C08666=1068.004,392.359,-109.873,175.287,34.758,156.445
C08667=1067.997,392.112,-109.833,175.281,34.751,156.443
C08668=1067.989,391.865,-109.792,175.276,34.743,156.441
C08669=1067.983,391.620,-109.751,175.271,34.735,156.440
C08670=1067.976,391.372,-109.711,175.266,34.727,156.438
C08671=1067.968,391.126,-109.670,175.261,34.720,156.436
C08672=1067.961,390.880,-109.629,175.256,34.712,156.434
C08673=1067.954,390.633,-109.589,175.252,34.705,156.433
C08674=1067.946,390.387,-109.548,175.246,34.697,156.431
C08675=1067.940,390.140,-109.508,175.242,34.690,156.429
C08676=1067.932,389.894,-109.467,175.236,34.682,156.428
C08677=1067.924,389.647,-109.427,175.231,34.675,156.426
C08678=1067.917,389.401,-109.386,175.226,34.667,156.424
C08679=1067.909,389.154,-109.347,175.221,34.660,156.423
C08680=1067.902,388.907,-109.306,175.217,34.652,156.421
C08681=1067.895,388.661,-109.266,175.211,34.645,156.419
C08682=1067.888,388.414,-109.225,175.207,34.637,156.417
C08683=1067.881,388.168,-109.186,175.201,34.630,156.416
C08684=1067.874,387.921,-109.144,175.197,34.622,156.414
C08685=1067.867,387.675,-109.105,175.192,34.615,156.412
C08686=1067.860,387.428,-109.064,175.187,34.608,156.411
C08687=1067.852,387.182,-109.025,175.182,34.600,156.409
C08688=1067.845,386.935,-108.985,175.177,34.593,156.407
C08689=1067.838,386.688,-108.945,175.172,34.586,156.406
C08690=1067.830,386.425,-108.902,175.167,34.578,156.404
C08691=1067.823,386.162,-108.858,175.162,34.570,156.402
C08692=1067.816,385.898,-108.816,175.157,34.562,156.401
C08693=1067.808,385.635,-108.773,175.151,34.555,156.399
C08694=1067.800,385.388,-108.733,175.147,34.547,156.397
C08695=1067.793,385.142,-108.694,175.142,34.540,156.396
C08696=1067.787,384.895,-108.654,175.138,34.533,156.394
C08697=1067.779,384.648,-108.614,175.132,34.526,156.392
C08698=1067.772,384.402,-108.574,175.128,34.519,156.391
C08699=1067.765,384.156,-108.534,175.123,34.512,156.389
C08700=1067.758,383.909,-108.494,175.118,34.504,156.388
C08701=1067.752,383.662,-108.455,175.113,34.497,156.386
C08702=1067.744,383.415,-108.415,175.109,34.490,156.384
C08703=1067.737,383.168,-108.375,175.105,34.483,156.383
C08704=1067.730,382.922,-108.335,175.099,34.476,156.381
C08705=1067.723,382.676,-108.296,175.095,34.469,156.380
C08706=1067.716,382.428,-108.256,175.090,34.462,156.378
C08707=1067.709,382.182,-108.216,175.086,34.455,156.376
C08708=1067.702,381.936,-108.177,175.080,34.448,156.375
C08709=1067.695,381.689,-108.138,175.076,34.441,156.373
C08710=1067.688,381.442,-108.098,175.071,34.434,156.372
C08711=1067.682,381.195,-108.058,175.067,34.427,156.370
C08712=1067.675,380.948,-108.019,175.062,34.420,156.369
C08713=1067.668,380.702,-107.980,175.057,34.413,156.367
C08714=1067.660,380.455,-107.940,175.053,34.406,156.366
C08715=1067.653,380.208,-107.901,175.048,34.399,156.364
C08716=1067.646,379.962,-107.862,175.043,34.392,156.363
C08717=1067.639,379.715,-107.823,175.039,34.386,156.361
C08718=1067.632,379.468,-107.783,175.034,34.379,156.360
C08719=1067.625,379.221,-107.744,175.030,34.372,156.358
C08720=1067.618,378.974,-107.705,175.025,34.365,156.356
C08721=1067.611,378.728,-107.666,175.020,34.358,156.355
C08722=1067.604,378.481,-107.627,175.016,34.351,156.354
C08723=1067.597,378.234,-107.588,175.011,34.345,156.352
C08724=1067.590,377.987,-107.549,175.007,34.338,156.351
C08725=1067.583,377.741,-107.509,175.002,34.331,156.349
C08726=1067.576,377.494,-107.471,174.998,34.324,156.348
C08727=1067.569,377.247,-107.432,174.993,34.318,156.346
C08728=1067.562,377.000,-107.393,174.988,34.311,156.345
C08729=1067.555,376.753,-107.354,174.984,34.305,156.343
C08730=1067.549,376.507,-107.315,174.980,34.298,156.342
C08731=1067.542,376.260,-107.276,174.975,34.291,156.340
C08732=1067.535,376.013,-107.237,174.971,34.284,156.339
C08733=1067.528,375.766,-107.199,174.966,34.278,156.337
C08734=1067.521,375.519,-107.159,174.962,34.271,156.336
C08735=1067.514,375.272,-107.121,174.957,34.265,156.334
C08736=1067.507,375.025,-107.082,174.952,34.258,156.333
C08737=1067.501,374.779,-107.043,174.948,34.252,156.332
C08738=1067.493,374.532,-107.005,174.944,34.245,156.330
C08739=1067.487,374.286,-106.966,174.939,34.238,156.329
C08740=1067.480,374.039,-106.927,174.935,34.232,156.327
C08741=1067.473,373.792,-106.889,174.931,34.225,156.326
C08742=1067.466,373.551,-106.851,174.926,34.219,156.324
C08743=1067.460,373.311,-106.814,174.922,34.213,156.323
C08744=1067.453,373.072,-106.776,174.918,34.206,156.322
C08745=1067.446,372.831,-106.738,174.913,34.200,156.320
C08746=1067.440,372.591,-106.701,174.909,34.194,156.319
C08747=1067.433,372.351,-106.664,174.905,34.188,156.318
C08748=1067.426,372.111,-106.627,174.900,34.181,156.316
C08749=1067.419,371.871,-106.589,174.896,34.175,156.315
C08750=1067.413,371.624,-106.551,174.892,34.169,156.314
C08751=1067.405,371.378,-106.512,174.887,34.162,156.312
C08752=1067.399,371.130,-106.474,174.883,34.156,156.311
C08753=1067.392,370.884,-106.436,174.879,34.150,156.309
C08754=1067.385,370.637,-106.398,174.875,34.143,156.308
C08755=1067.378,370.390,-106.359,174.870,34.137,156.307
C08756=1067.371,370.143,-106.322,174.866,34.131,156.305
C08757=1067.364,369.896,-106.283,174.862,34.125,156.304
C08758=1067.358,369.649,-106.245,174.857,34.118,156.303
C08759=1067.350,369.402,-106.207,174.853,34.112,156.301
C08760=1067.344,369.155,-106.169,174.849,34.106,156.300
C08761=1067.337,368.908,-106.131,174.844,34.100,156.299
C08762=1067.330,368.661,-106.093,174.840,34.093,156.297
C08763=1067.324,368.414,-106.054,174.836,34.087,156.296
C08764=1067.317,368.167,-106.017,174.832,34.081,156.294
C08765=1067.310,367.921,-105.978,174.827,34.075,156.293
C08766=1067.303,367.674,-105.941,174.823,34.068,156.292
C08767=1067.297,367.426,-105.903,174.819,34.062,156.290
C08768=1067.289,367.179,-105.865,174.814,34.056,156.289
C08769=1067.283,366.933,-105.827,174.810,34.050,156.288
C08770=1067.276,366.686,-105.789,174.806,34.044,156.286
C08771=1067.269,366.438,-105.751,174.802,34.038,156.285
C08772=1067.263,366.191,-105.713,174.797,34.031,156.284
C08773=1067.256,365.944,-105.676,174.793,34.025,156.282
C08774=1067.250,365.697,-105.638,174.790,34.019,156.281
C08775=1067.243,365.450,-105.601,174.786,34.013,156.280
C08776=1067.237,365.203,-105.562,174.781,34.007,156.279
C08777=1067.229,364.956,-105.525,174.777,34.001,156.277
C08778=1067.223,364.709,-105.487,174.773,33.995,156.276
C08779=1067.216,364.462,-105.450,174.768,33.989,156.275
C08780=1067.209,364.215,-105.412,174.764,33.983,156.273
C08781=1067.203,363.968,-105.374,174.760,33.977,156.272
C08782=1067.196,363.721,-105.337,174.756,33.971,156.271
C08783=1067.189,363.474,-105.299,174.751,33.965,156.270
C08784=1067.183,363.227,-105.262,174.747,33.959,156.268
C08785=1067.176,362.979,-105.225,174.744,33.953,156.267
C08786=1067.169,362.733,-105.188,174.740,33.947,156.266
C08787=1067.163,362.485,-105.149,174.735,33.941,156.264
C08788=1067.155,362.238,-105.112,174.731,33.935,156.263
C08789=1067.149,361.991,-105.075,174.727,33.930,156.262
C08790=1067.142,361.744,-105.038,174.723,33.923,156.261
C08791=1067.136,361.497,-105.000,174.719,33.917,156.259
C08792=1067.129,361.250,-104.963,174.714,33.912,156.258
C08793=1067.122,361.003,-104.926,174.711,33.906,156.257
C08794=1067.115,360.756,-104.889,174.707,33.900,156.256
C08795=1067.108,360.508,-104.852,174.703,33.894,156.254
C08796=1067.102,360.262,-104.814,174.698,33.888,156.253
C08797=1067.095,360.014,-104.777,174.694,33.882,156.252
C08798=1067.089,359.783,-104.742,174.691,33.877,156.251
C08799=1067.083,359.552,-104.707,174.687,33.872,156.250
C08800=1067.076,359.320,-104.673,174.683,33.866,156.249
C08801=1067.070,359.089,-104.638,174.679,33.861,156.247
C08802=1067.064,358.858,-104.604,174.675,33.855,156.246
C08803=1067.058,358.627,-104.569,174.672,33.850,156.245
C08804=1067.052,358.395,-104.535,174.668,33.844,156.244
C08805=1067.045,358.163,-104.500,174.665,33.839,156.243
C08806=1067.038,357.916,-104.463,174.660,33.834,156.242
C08807=1067.031,357.669,-104.427,174.656,33.828,156.240
C08808=1067.025,357.422,-104.389,174.652,33.822,156.239
C08809=1067.019,357.175,-104.353,174.648,33.816,156.238
C08810=1067.012,356.927,-104.316,174.645,33.811,156.237
C08811=1067.005,356.681,-104.279,174.640,33.805,156.236
C08812=1066.998,356.433,-104.242,174.636,33.800,156.235
C08813=1066.992,356.186,-104.206,174.632,33.794,156.233
C08814=1066.985,355.939,-104.169,174.628,33.788,156.232
C08815=1066.978,355.691,-104.132,174.625,33.783,156.231
C08816=1066.972,355.445,-104.095,174.620,33.777,156.230
C08817=1066.965,355.198,-104.059,174.616,33.771,156.229
C08818=1066.958,354.950,-104.022,174.612,33.765,156.227
C08819=1066.952,354.703,-103.986,174.609,33.760,156.226
C08820=1066.946,354.456,-103.949,174.605,33.754,156.225
C08821=1066.939,354.208,-103.912,174.601,33.749,156.224
C08822=1066.933,353.961,-103.876,174.596,33.743,156.223
C08823=1066.926,353.714,-103.839,174.593,33.738,156.222
C08824=1066.919,353.466,-103.803,174.589,33.732,156.220
C08825=1066.913,353.219,-103.766,174.585,33.727,156.219
C08826=1066.907,352.972,-103.730,174.581,33.721,156.218
C08827=1066.900,352.725,-103.693,174.577,33.716,156.217
C08828=1066.893,352.477,-103.656,174.573,33.710,156.216
C08829=1066.887,352.230,-103.620,174.569,33.705,156.215
C08830=1066.880,351.984,-103.584,174.566,33.699,156.213
C08831=1066.874,351.736,-103.548,174.562,33.694,156.212
C08832=1066.867,351.488,-103.512,174.558,33.688,156.211
C08833=1066.861,351.241,-103.475,174.554,33.683,156.210
C08834=1066.854,350.994,-103.439,174.550,33.677,156.209
C08835=1066.847,350.747,-103.403,174.546,33.672,156.208
C08836=1066.841,350.499,-103.367,174.542,33.666,156.207
C08837=1066.834,350.252,-103.330,174.539,33.661,156.206
C08838=1066.827,350.005,-103.295,174.535,33.655,156.204
C08839=1066.821,349.758,-103.259,174.531,33.650,156.203
C08840=1066.815,349.511,-103.222,174.527,33.645,156.202
C08841=1066.807,349.263,-103.186,174.523,33.639,156.201
C08842=1066.801,349.015,-103.150,174.519,33.634,156.200
C08843=1066.795,348.768,-103.114,174.516,33.629,156.199
C08844=1066.789,348.521,-103.078,174.512,33.623,156.198
C08845=1066.782,348.274,-103.042,174.508,33.618,156.197
C08846=1066.776,348.026,-103.007,174.504,33.612,156.195
C08847=1066.769,347.779,-102.970,174.500,33.607,156.194
C08848=1066.762,347.531,-102.935,174.496,33.602,156.193
C08849=1066.756,347.284,-102.898,174.493,33.597,156.192
C08850=1066.749,347.037,-102.863,174.489,33.591,156.191
C08851=1066.742,346.790,-102.827,174.486,33.586,156.190
C08852=1066.736,346.542,-102.791,174.482,33.581,156.189
C08853=1066.729,346.295,-102.755,174.478,33.576,156.188
C08854=1066.724,346.065,-102.722,174.474,33.570,156.187
C08855=1066.718,345.836,-102.689,174.471,33.566,156.186
C08856=1066.711,345.607,-102.656,174.467,33.560,156.185
C08857=1066.706,345.377,-102.623,174.464,33.556,156.184
C08858=1066.700,345.148,-102.589,174.461,33.551,156.183
C08859=1066.693,344.919,-102.557,174.457,33.546,156.182
C08860=1066.688,344.689,-102.523,174.454,33.541,156.181
C08861=1066.682,344.460,-102.490,174.451,33.537,156.180
C08862=1066.676,344.234,-102.458,174.446,33.532,156.179
C08863=1066.670,344.010,-102.425,174.443,33.527,156.178
C08864=1066.664,343.785,-102.393,174.440,33.522,156.177
C08865=1066.659,343.559,-102.361,174.437,33.517,156.176
C08866=1066.652,343.312,-102.326,174.433,33.512,156.175
C08867=1066.645,343.065,-102.290,174.429,33.507,156.174
C08868=1066.639,342.818,-102.254,174.426,33.502,156.173
C08869=1066.632,342.570,-102.219,174.422,33.497,156.172
C08870=1066.625,342.323,-102.184,174.419,33.492,156.171
C08871=1066.619,342.075,-102.148,174.414,33.487,156.170
C08872=1066.612,341.828,-102.113,174.411,33.482,156.169
C08873=1066.606,341.581,-102.078,174.407,33.476,156.168
C08874=1066.600,341.333,-102.042,174.403,33.471,156.166
C08875=1066.593,341.086,-102.007,174.400,33.466,156.166
C08876=1066.586,340.838,-101.972,174.396,33.461,156.164
C08877=1066.580,340.590,-101.936,174.393,33.456,156.163
C08878=1066.573,340.343,-101.901,174.389,33.451,156.162
C08879=1066.567,340.096,-101.866,174.386,33.446,156.161
C08880=1066.561,339.847,-101.831,174.381,33.440,156.160
C08881=1066.555,339.601,-101.796,174.378,33.436,156.159
C08882=1066.548,339.353,-101.761,174.374,33.430,156.158
C08883=1066.542,339.106,-101.725,174.371,33.426,156.157
C08884=1066.535,338.858,-101.690,174.367,33.420,156.156
C08885=1066.528,338.611,-101.655,174.364,33.415,156.155
C08886=1066.522,338.363,-101.621,174.360,33.410,156.154
C08887=1066.516,338.116,-101.585,174.357,33.405,156.153
C08888=1066.510,337.869,-101.550,174.353,33.400,156.152
C08889=1066.503,337.621,-101.515,174.350,33.395,156.151
C08890=1066.496,337.373,-101.481,174.346,33.390,156.150
C08891=1066.490,337.126,-101.445,174.342,33.385,156.149
C08892=1066.484,336.878,-101.410,174.338,33.380,156.148
C08893=1066.478,336.631,-101.376,174.335,33.375,156.147
C08894=1066.471,336.384,-101.341,174.331,33.370,156.146
C08895=1066.465,336.136,-101.306,174.328,33.366,156.145
C08896=1066.458,335.888,-101.271,174.324,33.360,156.144
C08897=1066.451,335.640,-101.237,174.321,33.356,156.143
C08898=1066.445,335.394,-101.202,174.317,33.350,156.142
C08899=1066.439,335.146,-101.167,174.314,33.346,156.141
C08900=1066.432,334.898,-101.132,174.310,33.341,156.140
C08901=1066.425,334.650,-101.098,174.307,33.336,156.139
C08902=1066.419,334.404,-101.063,174.304,33.331,156.138
C08903=1066.413,334.156,-101.029,174.300,33.326,156.137
C08904=1066.406,333.908,-100.994,174.296,33.322,156.136
C08905=1066.400,333.661,-100.959,174.292,33.316,156.135
C08906=1066.393,333.414,-100.924,174.289,33.312,156.134
C08907=1066.387,333.166,-100.890,174.285,33.307,156.133
C08908=1066.381,332.918,-100.856,174.282,33.301,156.132
C08909=1066.374,332.671,-100.821,174.279,33.297,156.131
C08910=1066.369,332.427,-100.787,174.275,33.292,156.130
C08911=1066.362,332.185,-100.753,174.272,33.287,156.129
C08912=1066.356,331.942,-100.719,174.268,33.282,156.128
C08913=1066.349,331.698,-100.686,174.265,33.278,156.127
C08914=1066.344,331.455,-100.651,174.262,33.273,156.126
C08915=1066.337,331.212,-100.618,174.258,33.268,156.126
C08916=1066.331,330.969,-100.584,174.255,33.264,156.125
C08917=1066.325,330.726,-100.551,174.252,33.259,156.124
C08918=1066.318,330.479,-100.516,174.248,33.254,156.123
C08919=1066.312,330.231,-100.482,174.244,33.249,156.122
C08920=1066.305,329.984,-100.448,174.241,33.245,156.121
C08921=1066.298,329.736,-100.413,174.237,33.240,156.120
C08922=1066.293,329.489,-100.379,174.234,33.235,156.119
C08923=1066.285,329.241,-100.345,174.230,33.230,156.118
C08924=1066.279,328.993,-100.311,174.227,33.226,156.117
C08925=1066.273,328.746,-100.277,174.224,33.221,156.116
C08926=1066.266,328.498,-100.243,174.220,33.216,156.115
C08927=1066.260,328.251,-100.209,174.217,33.212,156.114
C08928=1066.253,328.003,-100.175,174.213,33.207,156.113
C08929=1066.246,327.755,-100.141,174.210,33.202,156.112
C08930=1066.241,327.508,-100.107,174.207,33.198,156.111
C08931=1066.233,327.260,-100.073,174.203,33.193,156.111
C08932=1066.227,327.013,-100.039,174.200,33.188,156.110
C08933=1066.221,326.765,-100.005,174.197,33.183,156.109
C08934=1066.215,326.517,-99.972,174.193,33.179,156.108
C08935=1066.208,326.269,-99.937,174.190,33.175,156.107
C08936=1066.202,326.022,-99.904,174.187,33.170,156.106
C08937=1066.195,325.774,-99.869,174.183,33.165,156.105
C08938=1066.189,325.527,-99.835,174.180,33.160,156.104
C08939=1066.182,325.279,-99.802,174.177,33.156,156.103
C08940=1066.177,325.031,-99.768,174.172,33.151,156.102
C08941=1066.169,324.784,-99.734,174.169,33.147,156.101
C08942=1066.163,324.536,-99.700,174.166,33.142,156.100
C08943=1066.157,324.288,-99.667,174.162,33.137,156.099
C08944=1066.151,324.041,-99.633,174.159,33.132,156.099
C08945=1066.144,323.793,-99.599,174.156,33.128,156.098
C08946=1066.138,323.545,-99.566,174.152,33.123,156.097
C08947=1066.132,323.298,-99.532,174.149,33.119,156.096
C08948=1066.125,323.050,-99.498,174.146,33.114,156.095
C08949=1066.119,322.802,-99.465,174.143,33.110,156.094
C08950=1066.112,322.555,-99.431,174.139,33.105,156.093
C08951=1066.106,322.307,-99.397,174.136,33.100,156.092
C08952=1066.100,322.060,-99.364,174.133,33.095,156.091
C08953=1066.094,321.812,-99.330,174.129,33.091,156.090
C08954=1066.087,321.564,-99.297,174.126,33.086,156.089
C08955=1066.081,321.317,-99.263,174.123,33.082,156.089
C08956=1066.074,321.069,-99.230,174.120,33.077,156.088
C08957=1066.069,320.821,-99.196,174.116,33.073,156.087
C08958=1066.062,320.574,-99.163,174.113,33.068,156.086
C08959=1066.056,320.326,-99.129,174.110,33.064,156.085
C08960=1066.050,320.078,-99.096,174.107,33.059,156.084
C08961=1066.044,319.830,-99.063,174.103,33.054,156.083
C08962=1066.037,319.583,-99.029,174.100,33.050,156.082
C08963=1066.031,319.335,-98.995,174.097,33.045,156.081
C08964=1066.025,319.088,-98.962,174.094,33.040,156.080
C08965=1066.019,318.840,-98.929,174.090,33.036,156.080
C08966=1066.013,318.605,-98.898,174.087,33.031,156.079
C08967=1066.007,318.370,-98.865,174.084,33.027,156.078
C08968=1066.002,318.135,-98.834,174.081,33.023,156.077
C08969=1065.995,317.900,-98.803,174.078,33.019,156.076
C08970=1065.990,317.666,-98.771,174.075,33.015,156.075
C08971=1065.983,317.430,-98.739,174.072,33.010,156.074
C08972=1065.978,317.196,-98.708,174.069,33.006,156.074
C08973=1065.972,316.961,-98.677,174.066,33.001,156.073
C08974=1065.966,316.713,-98.643,174.063,32.997,156.072
C08975=1065.960,316.466,-98.610,174.060,32.993,156.071
C08976=1065.954,316.218,-98.577,174.056,32.988,156.070
C08977=1065.947,315.970,-98.543,174.053,32.983,156.069
C08978=1065.942,315.722,-98.510,174.050,32.979,156.068
C08979=1065.935,315.475,-98.477,174.047,32.974,156.067
C08980=1065.929,315.228,-98.444,174.044,32.970,156.067
C08981=1065.923,314.980,-98.411,174.040,32.965,156.066
C08982=1065.917,314.732,-98.378,174.037,32.961,156.065
C08983=1065.911,314.484,-98.344,174.034,32.956,156.064
C08984=1065.905,314.237,-98.312,174.031,32.952,156.063
C08985=1065.899,313.989,-98.279,174.028,32.947,156.062
C08986=1065.892,313.741,-98.246,174.024,32.943,156.061
C08987=1065.885,313.493,-98.213,174.021,32.939,156.061
C08988=1065.879,313.246,-98.180,174.018,32.934,156.060
C08989=1065.873,312.998,-98.148,174.015,32.930,156.059
C08990=1065.867,312.750,-98.115,174.012,32.925,156.058
C08991=1065.861,312.502,-98.083,174.009,32.921,156.057
C08992=1065.854,312.254,-98.050,174.005,32.917,156.056
C08993=1065.847,312.006,-98.017,174.002,32.912,156.055
C08994=1065.841,311.759,-97.984,173.999,32.908,156.055
C08995=1065.835,311.511,-97.952,173.996,32.904,156.054
C08996=1065.828,311.264,-97.919,173.993,32.899,156.053
C08997=1065.822,311.016,-97.887,173.989,32.895,156.052
C08998=1065.816,310.768,-97.855,173.986,32.890,156.051
C08999=1065.809,310.520,-97.822,173.983,32.886,156.050
C09000=1065.803,310.273,-97.789,173.980,32.882,156.050
C09001=1065.797,310.025,-97.756,173.977,32.878,156.049
C09002=1065.791,309.777,-97.724,173.974,32.873,156.048
C09003=1065.784,309.529,-97.691,173.971,32.869,156.047
C09004=1065.777,309.281,-97.659,173.967,32.864,156.046
C09005=1065.771,309.033,-97.627,173.964,32.860,156.045
C09006=1065.764,308.786,-97.594,173.961,32.856,156.045
C09007=1065.758,308.538,-97.562,173.958,32.852,156.044
C09008=1065.752,308.290,-97.530,173.955,32.848,156.043
C09009=1065.746,308.042,-97.497,173.952,32.843,156.042
C09010=1065.740,307.794,-97.465,173.949,32.839,156.041
C09011=1065.734,307.546,-97.432,173.945,32.834,156.040
C09012=1065.727,307.299,-97.400,173.942,32.830,156.040
C09013=1065.721,307.052,-97.368,173.939,32.826,156.039
C09014=1065.715,306.804,-97.336,173.936,32.822,156.038
C09015=1065.709,306.556,-97.303,173.933,32.817,156.037
C09016=1065.703,306.308,-97.271,173.930,32.813,156.036
C09017=1065.696,306.060,-97.239,173.927,32.808,156.035
C09018=1065.690,305.813,-97.207,173.924,32.804,156.035
C09019=1065.684,305.564,-97.175,173.921,32.800,156.034
C09020=1065.677,305.317,-97.142,173.917,32.796,156.033
C09021=1065.671,305.069,-97.110,173.914,32.791,156.032
C09022=1065.666,304.836,-97.080,173.911,32.787,156.031
C09023=1065.659,304.603,-97.049,173.909,32.783,156.031
C09024=1065.654,304.370,-97.019,173.906,32.779,156.030
C09025=1065.648,304.137,-96.989,173.903,32.775,156.029
C09026=1065.642,303.904,-96.959,173.900,32.771,156.028
C09027=1065.636,303.671,-96.929,173.897,32.767,156.028
C09028=1065.630,303.438,-96.899,173.894,32.763,156.027
C09029=1065.625,303.205,-96.868,173.891,32.759,156.026
C09030=1065.618,302.957,-96.836,173.888,32.754,156.025
C09031=1065.613,302.710,-96.805,173.885,32.750,156.024
C09032=1065.607,302.461,-96.773,173.882,32.746,156.024
C09033=1065.600,302.214,-96.740,173.879,32.742,156.023
C09034=1065.594,301.966,-96.709,173.876,32.737,156.022
C09035=1065.588,301.718,-96.676,173.873,32.733,156.021
C09036=1065.582,301.470,-96.645,173.870,32.729,156.020
C09037=1065.576,301.223,-96.612,173.867,32.725,156.019
C09038=1065.569,300.975,-96.581,173.865,32.721,156.019
C09039=1065.563,300.726,-96.549,173.862,32.716,156.018
C09040=1065.558,300.479,-96.517,173.859,32.712,156.017
C09041=1065.552,300.231,-96.485,173.856,32.708,156.016
C09042=1065.545,299.983,-96.454,173.853,32.704,156.015
C09043=1065.540,299.735,-96.422,173.850,32.699,156.014
C09044=1065.534,299.488,-96.389,173.847,32.695,156.014
C09045=1065.527,299.240,-96.358,173.844,32.690,156.013
C09046=1065.521,298.992,-96.326,173.841,32.686,156.012
C09047=1065.515,298.744,-96.294,173.838,32.682,156.011
C09048=1065.509,298.496,-96.262,173.835,32.678,156.010
C09049=1065.503,298.249,-96.231,173.832,32.673,156.010
C09050=1065.497,298.001,-96.199,173.829,32.669,156.009
C09051=1065.491,297.752,-96.167,173.826,32.665,156.008
C09052=1065.485,297.505,-96.136,173.823,32.661,156.007
C09053=1065.479,297.257,-96.104,173.820,32.656,156.006
C09054=1065.473,297.009,-96.072,173.817,32.652,156.006
C09055=1065.467,296.761,-96.041,173.814,32.648,156.005
C09056=1065.461,296.513,-96.010,173.811,32.644,156.004
C09057=1065.455,296.265,-95.978,173.808,32.639,156.003
C09058=1065.449,296.018,-95.947,173.805,32.636,156.002
C09059=1065.443,295.769,-95.915,173.802,32.631,156.002
C09060=1065.436,295.521,-95.883,173.799,32.627,156.001
C09061=1065.431,295.273,-95.852,173.796,32.623,156.000
C09062=1065.424,295.025,-95.821,173.794,32.619,155.999
C09063=1065.417,294.777,-95.790,173.791,32.614,155.998
C09064=1065.412,294.530,-95.758,173.788,32.611,155.998
C09065=1065.406,294.281,-95.727,173.785,32.606,155.997
C09066=1065.399,294.034,-95.696,173.782,32.602,155.996
C09067=1065.393,293.786,-95.664,173.779,32.598,155.995
C09068=1065.387,293.538,-95.633,173.776,32.594,155.995
C09069=1065.380,293.290,-95.602,173.773,32.590,155.994
